(* CODESYS project mem_workflowlib.library
   Author: Ronny Walther
   Placeholder: MEM_WorkflowLib
   Title: MEM_WorkflowLib
   Version: 1.0.0.42
   Company: ME

Project tree, tasks and I/O mapping:
  libraries: Tc2_Standard, * (Beckhoff Automation GmbH); Tc2_System, * (Beckhoff Automation GmbH); Tc2_Utilities, * (Beckhoff Automation GmbH)
  AdsInterface/
    DUTs/
      data type eCmdProcessing
      data type eSendCmdProcessing
      data type TdocCmd
      data type TdocCmd2
      data type TdocRes
      data type TdocRes2
      data type TdwCmd2
      data type TdwRes2
      data type TwCmd
      data type TwCmd2
      data type TwRes
      data type TwRes2
      data type TxCmdRes
      data type TxCmdRes2
      data type TxCmdRes2Double
    function block FB_docCMD_Handler_Base [ST]: M_EnableCmd, M_ExecuteCommand, M_FinishCommand, M_Log, M_ReceiveCommand, P_EnabledInternally
    function block FB_SendAdsDocCmd_Base [ST]: M_EnableCmd, M_SendCmd, M_SetLocalData, P_CommandState, P_EnabledInternally
    function block FB_wCMD_docCMD_Handler_Base2 [ST]: A_LogResChanges, M_EnableCmd, M_ExecuteCommand, M_FinishCommand, M_Log, M_ReceiveCommand, P_EnabledInternally
    function block FB_wCMD_Handler_Base [ST]: M_EnableCmd, M_ExecuteCommand, M_FinishCommand, M_Log, M_ReceiveCommand, P_EnabledInternally
    global variables GVL_AdsInterface
    global variables GVL_AdsInterface_ERROR_IDS
    function InitializeAds_Incoming [ST]
    function InitializeAds_Outgoing [ST]
  DocManagement/
    DUTs/
      data type eDocPositionIndex
      data type sDocEvent
      data type sDocument
      data type ST_Document
      data type ST_Document_AdditionalData
      data type ST_Document_Path
      data type ST_Document_Position
      data type ST_Document_Processing
    program DocManagement [ST]: M_CheckDocsInPrevLocation, M_FindDoc, M_GetDocArrayInformation, M_GetDocInfoById, M_Initialize, M_InsertNewDoc, M_InsertNewDoc2, M_RedirectDoc, M_RemoveAllDocs, M_RemoveDoc, M_ResetDocMng, M_SethPath, M_SetReleased, P_iArraySize
    program DocManagement_Ext [ST]: M_CheckDocsInPrevLocation, M_FindDoc, M_GetDocArrayInformation, M_GetDocInfoById, M_Initialize, M_InsertNewDoc, M_RedirectDoc, M_RemoveAllDocs, M_RemoveDoc, M_ResetDocMng, M_SethPath, M_SetReleased, P_iArraySize
    global variables GVL_DocManagement
    global variables GVL_DocManagement_ERROR_IDS
  ErrorManagement/
    DUTs/
      data type E_ErrorLevels
      data type E_ErrorTypes
      data type eErrorHandlingMode
      data type eErrorHandlingMode_1
      data type eErrorNotificationMode
      data type eErrorNotificationMode_1
      data type eErrorTypes
      data type sErrorMsg
      data type sSystemError
      data type sSystemErrorEvent
      data type ST_ErrorMsg
      data type ST_SystemError
      data type ST_SystemErrorEvent
      data type tErrorConstant
    program ErrorManagement [ST]: M_GetErrorArrayInformation, M_GetErrorInfo, M_Initialize, M_InsertNewError, M_RemoveAllErrors, M_RemoveError, M_ResetSysErrorMng, M_SendAllErrorOnce, M_SendEvents, M_SendSingleError, P_bHaveAllErrorsBeenSentAtLeastOnce, P_ErrorNotificationMode, P_tEventIntervall, M_CreateEvent, M_CreateLogData
    program ErrorManagement_Ext [ST]: M_GetErrorArrayInformation, M_GetErrorInfo, M_Initialize, M_InsertNewError, M_RemoveAllErrors, M_RemoveError, M_ResetSysErrorMng, M_SendAllErrorOnce, M_SendEvents, M_SendSingleError, P_bHaveAllErrorsBeenSentAtLeastOnce, P_ErrorNotificationMode, P_tEventIntervall, M_CreateEvent, M_CreateLogData
    function block FB_ErrorHandler_Base [ST]: M_ExecuteHandling_Automatic, M_ExecuteHandling_Continue, M_ExecuteHandling_Repeat, M_IsHandlingModeAllowed, M_ResetFb, M_SetHandling, P_bHandlingAvailable, P_wAllowedHandlingModes
    global variables GVL_ErrorManagement
    global variables GVL_ErrorManagement_ERROR_IDS
  EventManager/
    DUTs/
      data type eValueEventNotificationModes
      data type sInfoEvent
      data type sInfoMessage
      data type sInfoMessageObject
      data type sValueEvent
      data type sValueEventNotificationParameter
      data type sValueEventObject
  Logging/
    DUTs/
      data type E_LogModes
      data type eLogLevel
      data type eLogPrgStates
      data type sLogMsg
      data type sLogMsgObject
    global variables GVL_Logging
    global variables GVL_Logging_ERROR_IDS
    program Logging [ST]: Debug, Error, Fatal, Info, M_Initialize, P_bAllDataWritten, P_bResetMaxLogBufferOccupancyInPct, P_iMaxFileSizeKB, P_iMaxLogBufferOccupancyInPct, P_LogLevel, P_LogPrgState, P_nCurLogBufferOccupancyInPct, Trace, Warn, M_CheckTargetAccess, M_CreateLogString, M_DeleteFile, M_GenerateFilepath, M_GetNextLogMsgtoWrite, M_InsertLog, M_RenameFile, M_UpdateCurFileSize, M_UpdateFilePath, M_UpdateSysTimeVar
  Standard/
    DUTs/
      data type E_RETVALUE
      data type eFbStates
      data type sMethodState
      data type ST_MethodState
      data type ST_MethodState_AdditionalData
      data type T_RETVALUE
    function Dec [ST]
    function block FB_MethodState [ST]: bBusy, bDone, bError, bTimeout, ErrorId, ErrorMsg, GoDoneState, GoNextState, GoSpecificState, GoStartState, iStateVar, Reset
    function block FB_MethodState_Ext [ST]: bBusy, bDone, bError, bTimeout, ErrorId, ErrorMsg, ErrorType, GoDoneState, GoNextState, GoSpecificState, GoStartState, iStateVar, Reset, T_RetVal
    function block FB_MethodState_Ext_Data [ST]
    global variables GVL
    function Inc [ST]
    function IsValidPtr [ST]
    interface ITF_MethodState: bBusy, bDone, bError, ErrorMsg, GoDoneState, GoNextState, GoSpecificState, GoStartState, iStateVar, Reset
    interface ITF_MethodState_Ext: bBusy, bDone, bError, ErrorMsg, GoDoneState, GoNextState, GoSpecificState, GoStartState, iStateVar, Reset
    function Scale [ST]
    function Switch [ST]
  Version/
    global variables Global_Version
  WorkstationFsm/
    DUTs/
      data type eSubState
      data type eWsOperationType
      data type eWsStates
      data type sWsConfiguration
    function block FB_WsFsm_Base [ST]: A_DoTransition, FB_init, M_ThrowError, M_ERROR_DO, M_PAST_HANDLING_DO, M_PAST_HANDLING_ENTRY, M_PAST_HANDLING_EXIT, M_PRE_HANDLING_DO, M_PRE_HANDLING_ENTRY, M_PRE_HANDLING_EXIT, M_FinishCycle, M_ResetWs, M_ResolveErrorState, M_StartNewCycle, P_bDocInWs, P_CurState, P_iDocId, P_pCurDoc, P_tWsProcTimeout, M_CYCLE_FINISHED_DO, M_CYCLE_FINISHED_ENTRY, M_CYCLE_FINISHED_EXIT, M_ERROR_ENTRY, M_ERROR_EXIT, M_IDLE_DO, M_IDLE_ENTRY, M_IDLE_EXIT, M_INIT_WS_DO, M_INIT_WS_ENTRY, M_INIT_WS_EXIT, M_MASTER_SYSTEM_PROCESSING_DO, M_MASTER_SYSTEM_PROCESSING_ENTRY, M_MASTER_SYSTEM_PROCESSING_EXIT, M_WS_PROCESSING_INTO_ERROR
    global variables GVL_Statemachine_ERROR_IDS
    function InitializeWsFsm_Base [ST]
    interface ITF_WsFsm: M_ERROR_DO, M_PAST_HANDLING_DO, M_PAST_HANDLING_ENTRY, M_PAST_HANDLING_EXIT, M_PRE_HANDLING_DO, M_PRE_HANDLING_ENTRY, M_PRE_HANDLING_EXIT
  00000000-0000-0000-0000-000000000000|ReleaseNotes.txt
  ReleaseNotes.txt
*)

// AdsInterface/DUTs/eCmdProcessing
{attribute 'qualified_only'}
TYPE eCmdProcessing :
(
	_UNDEFINED 			:= 0,
	_RECEIVING			:= 1,
	_WAITING_FOR_START	:= 2,
	_EXECUTING			:= 3,
	_ABORTING			:= 4,
	_FINISHING			:= 5
)UINT;
END_TYPE

// AdsInterface/DUTs/eSendCmdProcessing
{attribute 'qualified_only'}
TYPE eSendCmdProcessing :
(
	_UNDEFINED 	:= 0,
	_IDLE		:= 1,
	_SENDING	:= 2,
	_STARTING	:= 3,
	_EXECUTING	:= 4,
	_DONE		:= 5
)UINT;
END_TYPE

// AdsInterface/DUTs/TdocCmd
{attribute 'qualified_only'}
TYPE TdocCmd :
	STRUCT
		Control: 		WORD;					// 0 = stop, 1 = receive, 2 = start				
		Version: 		WORD;					// 0 = not defined, > 0 = version of the instruction	
		Reserved: 		WORD;
		ParaCount1:		BYTE;					// count of ParaData / byte                             		
		ParaTyp1:		BYTE;
		ParaData1:		DWORD;
		ParaCount2:		BYTE;					// count of ParaData / byte                             		
		ParaTyp2:		BYTE;
		ParaData2:		ARRAY [0..24] OF WORD;	// data									
	END_STRUCT
END_TYPE

// AdsInterface/DUTs/TdocCmd2
{attribute 'qualified_only'}
TYPE TdocCmd2 :
	STRUCT
		Control: 		WORD;					// 0 = stop, 1 = receive, 2 = start				
		Version: 		WORD;					// 0 = not defined, > 0 = version of the instruction
		CmdDataLengthIn8Byte:	BYTE;			// data lenth = const = 7 * 8 byte = 56 byte = 28 words
		ResDataLengthIn8Byte:	BYTE;			// data lenth = const = 7 * 8 byte = 56 byte = 28 words	
	
		//  rest 56 byte
		ParaCount1:		BYTE;					// count of ParaData / byte                             		
		ParaTyp1:		BYTE;
		ParaData1:		DWORD;
		ParaCount2:		BYTE;					// count of ParaData / byte                             		
		ParaTyp2:		BYTE;
		ParaData2:		ARRAY [0..23] OF WORD;	// data									
	END_STRUCT
END_TYPE

// AdsInterface/DUTs/TdocRes
{attribute 'qualified_only'}
TYPE TdocRes :
	STRUCT
		Status: 		WORD;					// 0 = not defined, 1 = received, 2 = aktive started, 3 = aktive aborting, 4 = finnished ok, 5 = finished stopped, 6 = finished error   
		Error: 			WORD;					// 0 = not defined, > 0 = error no
		ErrorComp: 		WORD;
		ParaCount1:		BYTE;					// count of ParaData / byte                             		
		ParaTyp1:		BYTE;
		ParaData1:		DWORD;
		ParaCount2:		BYTE;					// count of ParaData / byte                             		
		ParaTyp2:		BYTE;
		ParaData2:		ARRAY [0..24] OF WORD;	// data		
	END_STRUCT
END_TYPE

// AdsInterface/DUTs/TdocRes2
{attribute 'qualified_only'}
TYPE TdocRes2 :
	STRUCT
		Status: 		WORD;					// 0 = not defined, 1 = received, 2 = aktive started, 3 = aktive aborting, 4 = finnished ok, 5 = finished stopped, 6 = finished error   
		Error: 			WORD;					// 0 = not defined, > 0 = error no
		ErrorComp: 		WORD;
		
		//  rest 56 byte
		ParaCount1:		BYTE;					// count of ParaData / byte                             		
		ParaTyp1:		BYTE;
		ParaData1:		DWORD;
		ParaCount2:		BYTE;					// count of ParaData / byte                             		
		ParaTyp2:		BYTE;
		ParaData2:		ARRAY [0..23] OF WORD;	// data		
	END_STRUCT
END_TYPE

// AdsInterface/DUTs/TdwCmd2
{attribute 'qualified_only'}
TYPE TdwCmd2 :
	STRUCT
		Control: 				WORD;					// 0 = stop, 1 = receive, 2 = start				
		Version: 				WORD;					// 0 = not defined, > 0 = version of the instruction	
		CmdDataLengthIn8Byte:	BYTE;					// data lenth = const = 7 * 8 byte = 56 byte = 28 words
		ResDataLengthIn8Byte:	BYTE;					// data lenth = const = 7 * 8 byte = 56 byte = 28 words	
		
		//  rest 56 byte
		ParaCount1:				BYTE;					// count of ParaData / byte                             		
		ParaTyp1:				BYTE;		
		ParaData1:				ARRAY [0..12] OF DWORD;	// data
		ParaDummy1:				WORD;									
	END_STRUCT
END_TYPE

// AdsInterface/DUTs/TdwRes2
{attribute 'qualified_only'}
TYPE TdwRes2 :
	STRUCT
		Status: 		WORD;					// 0 = not defined, 1 = received, 2 = aktive started, 3 = aktive aborting, 4 = finnished ok, 5 = finished stopped, 6 = finished error   
												// 4 = finnished ok, 5 = finished stopped, 6 = finished error  
		Error: 			WORD;					// Unique Error ID, see GVL_Error_Constants
		ErrorComp: 		WORD;					// Unique Component ID, see GVL_Error_Constants
		
		//  rest 56 byte
		ParaCount1:		BYTE;					// count of ParaData / byte                             		
		ParaTyp1:		BYTE;
		ParaData1:		ARRAY [0..12] OF DWORD;	// parameter field
		ParaDummy1:		WORD;
	END_STRUCT
END_TYPE

// AdsInterface/DUTs/TwCmd
{attribute 'qualified_only'}
TYPE TwCmd :
	STRUCT
		Control: 		WORD;					// 0 = stop, 1 = receive, 2 = start				
		Version: 		WORD;					// 0 = not defined, > 0 = version of the instruction	
		Reserved: 		WORD;
		ParaCount:		BYTE;					// count of ParaData / byte                             		
		ParaTyp:		BYTE;
		ParaData:		ARRAY [0..27] OF WORD;	// data									
	END_STRUCT
END_TYPE

// AdsInterface/DUTs/TwCmd2
{attribute 'qualified_only'}
TYPE TwCmd2 :
	STRUCT
		Control: 				WORD;					// 0 = stop, 1 = receive, 2 = start				
		Version: 				WORD;					// 0 = not defined, > 0 = version of the instruction	
		CmdDataLengthIn8Byte:	BYTE;					// data lenth = const = 7 * 8 byte = 56 byte = 28 words
		ResDataLengthIn8Byte:	BYTE;					// data lenth = const = 7 * 8 byte = 56 byte = 28 words	
		
		//  rest 56 byte
		ParaCount1:				BYTE;					// count of ParaData / byte                             		
		ParaTyp1:				BYTE;		
		ParaData1:				ARRAY [0..26] OF WORD;	// data									
	END_STRUCT
END_TYPE

// AdsInterface/DUTs/TwRes
{attribute 'qualified_only'}
TYPE TwRes :
	STRUCT
		Status: 		WORD;					// 0 = not defined, 1 = received, 2 = aktive started, 3 = aktive aborting, 4 = finnished ok, 5 = finished stopped, 6 = finished error   
												// 4 = finnished ok, 5 = finished stopped, 6 = finished error  
		Error: 			WORD;					// Unique Error ID, see GVL_Error_Constants
		ErrorComp: 		WORD;					// Unique Component ID, see GVL_Error_Constants
		ParaCount:		BYTE;					// count of ParaData / byte                             		
		ParaTyp:		BYTE;
		ParaData:		ARRAY [0..27] OF WORD;	// parameter field
	END_STRUCT
END_TYPE

// AdsInterface/DUTs/TwRes2
{attribute 'qualified_only'}
TYPE TwRes2 :
	STRUCT
		Status: 		WORD;					// 0 = not defined, 1 = received, 2 = aktive started, 3 = aktive aborting, 4 = finnished ok, 5 = finished stopped, 6 = finished error   
												// 4 = finnished ok, 5 = finished stopped, 6 = finished error  
		Error: 			WORD;					// Unique Error ID, see GVL_Error_Constants
		ErrorComp: 		WORD;					// Unique Component ID, see GVL_Error_Constants
		
		//  rest 56 byte
		ParaCount1:		BYTE;					// count of ParaData / byte                             		
		ParaTyp1:		BYTE;
		ParaData1:		ARRAY [0..26] OF WORD;	// parameter field
	END_STRUCT
END_TYPE

// AdsInterface/DUTs/TxCmdRes
TYPE TxCmdRes :
	UNION
		wCmd: TwCmd;		// data of type word
		docCmd: TdocCmd;	// doc data type
		wRes: TwRes;		// data of type word
		docRes:	TdocRes;	// doc data type
	END_UNION
END_TYPE

// AdsInterface/DUTs/TxCmdRes2
TYPE TxCmdRes2 :
	UNION
		wCmd: TwCmd2;		// data of type word
		dwCmd: TdwCmd2;		// data of type dword
		docCmd: TdocCmd2;	// doc data type
		
		wRes: TwRes2;		// data of type word
		dwRes: TdwRes2;		// data of type dword
		docRes:	TdocRes2;	// doc data type
	END_UNION
END_TYPE

// AdsInterface/DUTs/TxCmdRes2Double
{attribute 'qualified_only'}
TYPE TxCmdRes2Double :
	STRUCT
		Cmd: TxCmdRes2;
		Res: TxCmdRes2;
	END_STRUCT
END_TYPE

// DocManagement/DUTs/eDocPositionIndex
TYPE eDocPositionIndex :
(
	UNDEFINED 	:= 0,
	POSITION_1 	:= 1,
	POSITION_2 	:= 2
)UINT;
END_TYPE

// DocManagement/DUTs/sDocEvent
//Event structure to send document tracking information without special request from host
//e.g. DocIn/ DocOut when entering/leaving a workstation and DocProcessStart when a doc is set to "UNRELEASED"
//Size: 6 Byte
TYPE sDocEvent :
	STRUCT
		DocID :				UDINT;	//Unique document id
		EventChangeFlag :	BOOL;	//assures that events ALWAYS differ from the previous one, not evaluated by host
	END_STRUCT
END_TYPE

// DocManagement/DUTs/sDocument
 
TYPE sDocument :
	STRUCT
		Free :					BOOL;	//0: Occupied, 1: Free
		ID :					UDINT;	//0: Document Identification (in the Machine)
		Module :				UINT;	//0: Invalid, 1: Modul 1, 2: Modul 2, 3: Modul 3
		Location :				UINT;	//0: Invalid, 1: RFID1, 2: RFID2, etc.
		Path :					UINT;	//Paths that the document could go through in the machine
		RedAtLocation :			UINT;	//0: No redirect, > 0: Location where document should be redirected
		RedToLocation :			UINT;	//0: No redirect, > 0: Location to where document should be redirected
		PositionIndex : 		UINT;	//Doc Position within a double usage. Only interesting if 2 different step sizes and 2 different layouts
		Released :				BOOL;	//0: Blocked, 1: Released (can be moved to next Location or picked up)
		bReleaseHandshakeActive: BOOL;	//Flag to switch release handshaking inside a non-virtual on or off
		Moving :				BOOL;	//0: Not Moving, 1: Moving
		bLockedBySps :			BOOL;	//FALSE: Doc can be modified by host, TRUE: Doc is locked by SPS and can not be modified by host
		Error :					BOOL;	//0: No Error, 1: Error
		//ErrorID :				WORD;	//ErrorID
	END_STRUCT
END_TYPE

// DocManagement/DUTs/ST_Document
 
TYPE ST_Document :
	STRUCT
		ID                      : UDINT;						//Unique document identification (in the Machine)

		stPosition 				: ST_Document_Position;			//Specifies the current position of the document inside the machine	
		stPath 					: ST_Document_Path; 			//Path of the document through the machine				
		stAdditionalData 		: ST_Document_AdditionalData;	//Various additional data
		stProcessing 			: ST_Document_Processing;		
		Free 					: BOOL;	//0: Occupied, 1: Free
	END_STRUCT
END_TYPE

// DocManagement/DUTs/ST_Document_AdditionalData
TYPE ST_Document_AdditionalData :
STRUCT
	DataString 	: STRING(GVL_DocManagement.MAX_INFO_TEXT_SIZE);
	DataField1	: LREAL;	//8bytes
	DataFiled2	: UDINT;	//4bytes
	DataField3	: UINT;		//2bytes
	DataField4 	: BYTE;		//1byte
END_STRUCT
END_TYPE

// DocManagement/DUTs/ST_Document_Path
TYPE ST_Document_Path :
STRUCT
		Path :					UINT;	//Paths that the document could go through in the machine
		RedAtLocation :			UINT;	//0: No redirect, > 0: Location where document should be redirected
		RedToLocation :			UINT;	//0: No redirect, > 0: Location to where document should be redirected
END_STRUCT
END_TYPE

// DocManagement/DUTs/ST_Document_Position
TYPE ST_Document_Position :
STRUCT		
		Module :				UINT;	//0: Invalid, 1: Modul 1, 2: Modul 2, 3: Modul 3
		Location :				UINT;	//0: Invalid, 1: RFID1, 2: RFID2, etc.
END_STRUCT
END_TYPE

// DocManagement/DUTs/ST_Document_Processing
TYPE ST_Document_Processing :
STRUCT
	bReleaseHandshakeActive	: BOOL;	//Flag to switch release handshaking inside a non-virtual on or off		
	Released 				: BOOL;	//0: Blocked, 1: Released (can be moved to next Location or picked up)	
	bLockedBySps 			: BOOL;	//FALSE: Doc can be modified by host, TRUE: Doc is locked by SPS and can not be modified by host
	Error 					: BOOL;	//FALSE: No Error, TRUE: Error
END_STRUCT
END_TYPE

// ErrorManagement/DUTs/E_ErrorLevels
{attribute 'qualified_only'}
TYPE E_ErrorLevels :
(
	_UNDEFINED 	:= 0,
	_WARNING	:= 1, 	//Machine continues running with some functionality deactivated eventually
	_ERROR		:= 2, 	//Machine shall be in ERROR state. Error can be solved by operator. A document reject could be possible
	_FATAL 		:= 3	//Machine shall be in ERROR state. Error can not be solved without major action. Could be a complete restart with all documents getting rejected
)UINT;
END_TYPE

// ErrorManagement/DUTs/E_ErrorTypes
{attribute 'qualified_only'}
TYPE E_ErrorTypes :
(
	SPS			:= 0, 	//firmware internal errors
	TWINCAT		:= 1 	//forwarded Beckhoff Twincat errors
)UINT;
END_TYPE

// ErrorManagement/DUTs/eErrorHandlingMode
{attribute 'qualified_only'}
TYPE eErrorHandlingMode :
(
	_NONE 		:= 0,
	_AUTOMATIC	:= 1,
	_REPEAT		:= 2,
	_CONTINUE	:= 3,
	_CANCEL		:= 4
)UINT;
END_TYPE

// ErrorManagement/DUTs/eErrorHandlingMode_1
{attribute 'qualified_only'}
TYPE eErrorHandlingMode_1 :
(
	_NONE 		:= 0,
	_AUTOMATIC	:= 1,
	_REPEAT		:= 2,
	_CONTINUE	:= 3,
	_CANCEL		:= 4
)UINT;
END_TYPE

// ErrorManagement/DUTs/eErrorNotificationMode
{attribute 'qualified_only'}
TYPE eErrorNotificationMode :
(
	UNDEFINED 							:= 0,
	SENDING_ERRORS_OFF					:= 1,
	SENDING_ERRORS_ONCE_IMMEDIATLY		:= 2,
	SENDING_ERRORS_ALWAYS_PERIODICALLY	:= 3
)UINT;
END_TYPE

// ErrorManagement/DUTs/eErrorNotificationMode_1
{attribute 'qualified_only'}
TYPE eErrorNotificationMode_1 :
(
	UNDEFINED 							:= 0,
	SENDING_ERRORS_OFF					:= 1,
	SENDING_ERRORS_ONCE_IMMEDIATLY		:= 2,
	SENDING_ERRORS_ALWAYS_PERIODICALLY	:= 3
)UINT;
END_TYPE

// ErrorManagement/DUTs/eErrorTypes
{attribute 'qualified_only'}
TYPE eErrorTypes :
(
	_UNDEFINED 	:= 0,
	_WARNING	:= 1, 	//Machine continues running with some functionality deactivated eventually
	_ERROR		:= 2, 	//Machine shall be in ERROR state. Error can be solved by operator. A document reject could be possible
	_FATAL 		:= 3	//Machine shall be in ERROR state. Error can not be solved without major action. Could be a complete restart with all documents getting rejected
)UINT;
END_TYPE

// ErrorManagement/DUTs/sErrorMsg
{attribute 'qualified_only'}
TYPE sErrorMsg : //to hold all SPS internal error messages
STRUCT
	//Categorization
		ErrorTyp : 		eErrorTypes;        //Undefined, Minor, Major, Fatal
	
	//Cause
		wModule : 		WORD := 1;				//Module no if redundant modules exist
		wComponent : 	WORD := 0;				//ID for each component
		wErrorNo : 		WORD := GVL.ERR_NO_ERROR;	//Error no (see GVL_Error_Constants)
		sFunctionName : STRING;					//name of (FSM) funtion which threw the error
	
	//Handling
		iRelatedDocId : UDINT := 0;
		pErrorHandler : POINTER TO FB_ErrorHandler_Base; //Pointer to specific error handler, if null pointer => no error handling
END_STRUCT
END_TYPE

// ErrorManagement/DUTs/sSystemError
{attribute 'qualified_only'}
TYPE sSystemError :
	STRUCT
		SysErrorMessageID :	UINT;		//Unique ID generated automatically by SysErrorMng. Helps to identify errors between SPS and host		
		ErrorMsg :			sErrorMsg;	//error msg structure
		bErrorWasSent :		BOOL;		//flag to indicate wether error was sent already or not
	END_STRUCT
END_TYPE

// ErrorManagement/DUTs/sSystemErrorEvent
//Event structure to send error information without special request from host
//Size: 18 Byte
{attribute 'qualified_only'}
TYPE sSystemErrorEvent :
	STRUCT
		iRelatedDocId : 		UDINT;			//rom error affected document, 0 = No doc affected
		
		SysErrorMessageID :		UINT;			//Unique ID generated automatically by SysErrorMng. Helps to identify errors between SPS and host
		
		ErrorTyp : 				eErrorTypes;	//Undefined, Minor, Major, Fatal		
		ErrorModuleId :			WORD;			//Machine module which holds the error reporting component	
		ErrorCompId :			WORD;			//Error reporting component
		ErrorId :				WORD;			//Unique error ID specifies the error happened

		AvailableHandlingModes:	WORD;			//Bits 0: none, 1:Automatic, 2:Repeat, 3: Continue
		EventChangeFlag:		BOOL;			//assures that events ALWAYS differ from the previous one, not evaluated by host
	END_STRUCT
END_TYPE

// ErrorManagement/DUTs/ST_ErrorMsg
{attribute 'qualified_only'}
TYPE ST_ErrorMsg : //to hold all SPS internal error messages
STRUCT
	//Categorization
		eErrorType : 		E_ErrorTypes; 
		eErrorLevel : 		E_ErrorLevels;        //Undefined, Minor, Major, Fatal
	
	//Cause
		wModule : 		WORD := 1;				//Module no if redundant modules exist
		wComponent : 	WORD := 0;				//ID for each component
		wErrorNo : 		WORD := GVL.ERR_NO_ERROR;	//Error no (see GVL_Error_Constants)
		sFunctionName : STRING;					//name of (FSM) funtion which threw the error
	
	//Handling
		iRelatedDocId : UDINT := 0;
		pErrorHandler : POINTER TO FB_ErrorHandler_Base; //Pointer to specific error handler, if null pointer => no error handling
END_STRUCT
END_TYPE

// ErrorManagement/DUTs/ST_SystemError
{attribute 'qualified_only'}
TYPE ST_SystemError :
	STRUCT
		SysErrorMessageID :	UINT;		//Unique ID generated automatically by SysErrorMng. Helps to identify errors between SPS and host		
		ErrorMsg :			ST_ErrorMsg;	//error msg structure
		bErrorWasSent :		BOOL;		//flag to indicate wether error was sent already or not
	END_STRUCT
END_TYPE

// ErrorManagement/DUTs/ST_SystemErrorEvent
//Event structure to send error information without special request from host
//Size: 18 Byte
{attribute 'qualified_only'}
TYPE ST_SystemErrorEvent :
	STRUCT
		iRelatedDocId : 		UDINT;			//rom error affected document, 0 = No doc affected
		
		SysErrorMessageID :		UINT;			//Unique ID generated automatically by SysErrorMng. Helps to identify errors between SPS and host
		
		ErrorTyp : 				E_ErrorLevels;	//Undefined, Minor, Major, Fatal		
		ErrorModuleId :			WORD;			//Machine module which holds the error reporting component	
		ErrorCompId :			WORD;			//Error reporting component
		ErrorId :				WORD;			//Unique error ID specifies the error happened

		AvailableHandlingModes:	WORD;			//Bits 0: none, 1:Automatic, 2:Repeat, 3: Continue
		EventChangeFlag:		BOOL;			//assures that events ALWAYS differ from the previous one, not evaluated by host
	END_STRUCT
END_TYPE

// ErrorManagement/DUTs/tErrorConstant
{attribute 'qualified_only'}
TYPE tErrorConstant : WORD (0..32767); END_TYPE
//Value is limited to 15bit because of ADS ME host connection DLL

// EventManager/DUTs/eValueEventNotificationModes
TYPE eValueEventNotificationModes :
(
	UNDEFINED 								:= 0,
	ON_CHANGE_ALWAYS						:= 1,
	ON_CHANGE_TIME_VALUE_DIFF_FROM_LAST		:= 2,
	ON_CHANGE_TIME_VALUE_DIFF_FROM_SPECIFIC	:= 3,
	ON_CHANGE_TIME							:= 4,
	TIME_CHANGE								:= 5
)UINT;
END_TYPE

// EventManager/DUTs/sInfoEvent
//Event structure to send general information without special request from host
//e.g. machine information, while performing some asynchrone action inside SPS
//Size: 6 Byte
TYPE sInfoEvent :
	STRUCT
		ComponentId :		WORD;	//Unique ID to identify the component the message came from
		InfoMessageId :		WORD;	//see GVL_Constants for pre-defined messages
		EventChangeFlag :	BOOL;	//assures that events ALWAYS differ from the previous one, not evaluated by host
	END_STRUCT
END_TYPE

// EventManager/DUTs/sInfoMessage
TYPE sInfoMessage :
STRUCT
	wComponentId :		WORD;	//Unique ID to identify the component the message came from
	wInfoMessageId :	WORD;	//see GVL_Constants for pre-defined messages
END_STRUCT
END_TYPE

// EventManager/DUTs/sInfoMessageObject
TYPE sInfoMessageObject :
STRUCT
	bEventIsValid	: BOOL;
	InfoMessage 	: sInfoMessage;
END_STRUCT
END_TYPE

// EventManager/DUTs/sValueEvent
TYPE sValueEvent : 
	STRUCT
		Value 			: WORD; //event specific value
		EventChangeFlag : BOOL;	//assures that events ALWAYS differ from the previous one, not evaluated by host
		 {attribute 'hide'}
		_reserved1 : USINT;
	END_STRUCT
END_TYPE

// EventManager/DUTs/sValueEventNotificationParameter
TYPE sValueEventNotificationParameter :
STRUCT
	NotificationMode 	: eValueEventNotificationModes;	//notification mode
	tSendInterval 		: TIME;							//Minimum send interval 
	iValueDiff			: UINT;							//trigger tolerance in Modes: ON_CHANGE_TIME_VALUE_DIFF_FROM_LAST and ON_CHANGE_TIME_VALUE_DIFF_FROM_SPECIFIC
	iSpecificRefValue	: UINT;							//reference value to be compared to in Mode: ON_CHANGE_TIME_VALUE_DIFF_FROM_SPECIFIC
END_STRUCT
END_TYPE

// EventManager/DUTs/sValueEventObject
TYPE sValueEventObject :
STRUCT
	bEventIsValid			: BOOL;
	strEventName			: STRING;
	pInternallyLinkedValue	: POINTER TO UINT;	
	pEvent 					: POINTER TO sValueEvent;
	EventParameter			: sValueEventNotificationParameter;
	tTimer					: TON;
END_STRUCT
END_TYPE

// Logging/DUTs/E_LogModes
{attribute 'qualified_only'}
{attribute 'strict'}
TYPE E_LogModes :
(
	KeepAllFiles 	:= 0,
	KeepTwoFiles 	:= 1
);
END_TYPE

// Logging/DUTs/eLogLevel
// ALL → TRACE → DEBUG → INFO → WARN → ERROR → FATAL → OFF.
{attribute 'qualified_only'}
TYPE eLogLevel :
(
	OFF			:= 0,	
//Log levels	
	FATAL		:= 1,
	ERROR 		:= 2,
	WARN 		:= 3,
	INFO 		:= 4,	
	DEBUG 		:= 5,
	TRACE		:= 6,	
	ALL			:= 7
)UINT;
END_TYPE

// Logging/DUTs/eLogPrgStates
{attribute 'qualified_only'}
TYPE eLogPrgStates :
(
	LOG_INITIALIZING 	:= 0,
	LOG_STAND_BY		:= 1,
	LOG_OPENING_FILE	:= 2,
	LOG_WRITING_FILE	:= 3,
	LOG_CLOSING_FILE	:= 4,
	LOG_ERROR			:= 5
)UINT;
END_TYPE

// Logging/DUTs/sLogMsg
{attribute 'qualified_only'}
TYPE sLogMsg :
	STRUCT
		LogLevel 			: eLogLevel;
		sCallFunctionName 	: STRING;			//name of (FSM) funtion which threw the error		
		sLogMessage 		: STRING(255);	
	END_STRUCT
END_TYPE

// Logging/DUTs/sLogMsgObject
{attribute 'hide'}
{attribute 'qualified_only'}
TYPE sLogMsgObject :
	STRUCT
		bIsValidMsg	: BOOL;
		iLogMsgId 	: UDINT;			//Unique ID generated automatically by SysErrorMng. Helps to identify errors between SPS and host
		sTimeStamp 	: STRING;
		LogMsg 		: sLogMsg;
	END_STRUCT
END_TYPE

// Standard/DUTs/E_RETVALUE
//{attribute 'qualified_only'}
//{attribute 'strict'}
TYPE E_RETVALUE :
(
	eOK 	 := 1,
	eBUSY 	 := 0,
	eNOK 	 := -1	
)INT;
END_TYPE

// Standard/DUTs/eFbStates
{attribute 'qualified_only'}
TYPE eFbStates : //Types to structure FB state machines
(
	_ENTRY 			:= 0,
	_OFF			:= 1,
	_POWERING_ON	:= 2,
	_INITIALIZING	:= 3,
	_IDLE			:= 4,
	_RUNNING		:= 5,
	_POWERING_OFF	:= 6,
	_ERROR			:= 7,	 
	_EXIT			:= 8
)uint;
END_TYPE

// Standard/DUTs/sMethodState
{attribute 'qualified_only'}
TYPE sMethodState :
STRUCT
	//Status flags
		bDone 		: BOOL;
		bError 		: BOOL;
		bBusy		: BOOL;
		(*
	//signals, if the corresponding status flag just changed (rising or falling edge)
		bDoneEdge,
		bErrorEdge,
		bBusyEdge	: BOOL;
		*)
	iStateVar	: UINT;
	ErrorMsg 	: sErrorMsg;
END_STRUCT
END_TYPE

// Standard/DUTs/ST_MethodState
{attribute 'qualified_only'}
TYPE ST_MethodState :
STRUCT
	//Status flags
		bDone 		: BOOL;
		bError 		: BOOL;
		bBusy		: BOOL;
		(*
	//signals, if the corresponding status flag just changed (rising or falling edge)
		bDoneEdge,
		bErrorEdge,
		bBusyEdge	: BOOL;
		*)
		iStateVar	: UINT;
		ErrorMsg 	: ST_ErrorMsg;
END_STRUCT
END_TYPE

// Standard/DUTs/ST_MethodState_AdditionalData
TYPE ST_MethodState_AdditionalData :
STRUCT
	DataString 	: STRING(GVL_DocManagement.MAX_INFO_TEXT_SIZE);
	DataField1	: LREAL;	//8bytes
	DataFiled2	: UDINT;	//4bytes
	DataField3	: UINT;		//2bytes
	DataField4 	: BYTE;		//1byte
END_STRUCT
END_TYPE

// Standard/DUTs/T_RETVALUE
TYPE T_RETVALUE : E_RETVALUE; END_TYPE

// WorkstationFsm/DUTs/eSubState
{attribute 'qualified_only'}
{attribute 'strict'}
TYPE eSubState :
(
	UNDEFINED 	:= 0,
	STATE_ENTRY	:= 1,
	STATE_DO	:= 2,
	STATE_EXIT	:= 3	
);
END_TYPE

// WorkstationFsm/DUTs/eWsOperationType
TYPE eWsOperationType :
(
	_UNDEFINED 				:= 0,
	_STEP_BY_STEP			:= 1,	//workstation cycling is controlled step by step
	_CONTINOUS_BY_TRIGGER	:= 2	//workstation cycling is triggered by a external s signal
)UINT;
END_TYPE

// WorkstationFsm/DUTs/eWsStates
TYPE eWsStates : //Possible Workstation states inside FB_WsFsm
(
	UNDEFINED 					:= 0,
	INIT_WS						:= 1,
	IDLE						:= 2,	//WS ready to be startet
	WS_PROCESSING				:= 3,	//WS running (including Master system processing)
	PRE_HANDLING				:= 4,	//optional code can be processed here
	MASTER_SYSTEM_PROCESSING	:= 5,	//Master system is processing the document
	PAST_HANDLING				:= 6,	//optional code can be processed here
	ERROR						:= 7,	//Ws in error
	CYCLE_FINISHED				:= 8	//Cycle ready to be finished
)UINT;
END_TYPE

// WorkstationFsm/DUTs/sWsConfiguration
TYPE sWsConfiguration :
STRUCT
	iWsNum : 					UINT;
	iRelDocNum :				UINT;	//Distance between previous and this WS in mm - 0 is OFF
	iLocation :					UINT;		
	bVirtualWs : 				BOOL;
	tWsProcessingTimeout :		TIME;	//Timeout for composite state WsProcessing
	OperationType: 				eWsOperationType;

//Doc events	
	pEvt_DocIn, 
	pEvt_DocProcessStart,
	pEvt_DocOut : 				POINTER TO sDocEvent;
	bEvt_DocIn_WasSet, 									//DocIn event set status
	pEvt_DocProcessStart_WasSet,						//DocProcessStart event set status
	pEvt_DocOut_wasSet 				: BOOL := FALSE;	//DocOut event set status
	
	wCompId : 					WORD;	
	//Document will be unlocked when method M_FinishCycle is called. 
	//Flag shall be set to TRUE, if Ws is the last WS to enable the host to remove the doc from the buffer
	bUnlockDocAtFinishing : BOOL; 
END_STRUCT
END_TYPE

// AdsInterface/GVL_AdsInterface
{attribute 'hide'}
{attribute 'qualified_only'}
VAR_GLOBAL
	wCompId_IncomingAds,
	wCompId_OutgoingAds 		: tErrorConstant	:= 0;
	
	wErrorIdOffset_IncomingAds,
 	wErrorIdOffset_OutgoingAds	: tErrorConstant	:= 0;
	
	bLoggingOnOff_IncomingAds,
	bLoggingOnOff_OutgoingAds 	: BOOL				:= FALSE;
END_VAR

// AdsInterface/GVL_AdsInterface_ERROR_IDS
{attribute 'qualified_only'}
VAR_GLOBAL CONSTANT	
	ERR_ITF_INCOMING_COMMAND_HAS_WRONG_VERSION :							tErrorConstant := 1;
	ERR_ITF_INCOMING_COMMAND_HAS_WRONG_PARAMETER_COUNT :					tErrorConstant := 2;
	ERR_ITF_INCOMING_COMMAND_HAS_WRONG_PARAMETER_TYP :						tErrorConstant := 3;
	ERR_ITF_INCOMING_COMMAND_IS_BLOCKED :									tErrorConstant := 4;
	ERR_ITF_COMMAND_CAN_NOT_BE_ENABLED_THUS_INTERNALLY_DISABLED:			tErrorConstant := 5;
	ERR_ITF_COMMAND_CAN_NOT_BE_ENABLED_THUS_EXTERNALLY_DISABLED:			tErrorConstant := 6;
	ERR_ITF_WRONG_COMMAND_DATA:												tErrorConstant := 7;
	ERR_ITF_COMMAND_EXECUTION_TIMEOUT:										tErrorConstant := 8;
	ERR_ITF_INCOMING_COMMAND_HAS_WRONG_COMMAND_DATA_SIZE:					tErrorConstant := 9;
	ERR_ITF_INCOMING_COMMAND_HAS_WRONG_RESULT_DATA_SIZE:					tErrorConstant := 10;
	
	ERR_ITF_COMMAND_WAS_ABORTED_BY_HOST_DURING_EXECUTION:					tErrorConstant := 15;

	//ADS Sending errors
	ERR_ITF_WRONG_FB_STATE_TO_SEND_COMMAND :								tErrorConstant := 50;
	
END_VAR

// DocManagement/GVL_DocManagement
{attribute 'qualified_only'}
{attribute 'hide'}
VAR_GLOBAL
	wCompId 					: tErrorConstant	:= 0;
	wErrorIdOffset 				: tErrorConstant	:= 0;
END_VAR
VAR_GLOBAL CONSTANT
	MAX_INFO_TEXT_SIZE 			: UINT 				:= 50; 
END_VAR

// DocManagement/GVL_DocManagement_ERROR_IDS
{attribute 'qualified_only'}
VAR_GLOBAL CONSTANT
	
	ERR_DOC_ID_NOT_FOUND :													tErrorConstant := 2;
	ERR_DOC_ARRAY_FULL : 													tErrorConstant := 3;
	ERR_DOC_CAN_NOT_BE_INSERTED_THUS_DOC_ID_EXISTENT_ALREADY :				tErrorConstant := 4;
	ERR_DOC_CAN_NOT_BE_INSERTED_THUS_ARRAY_FULL :							tErrorConstant := 5;
	
	ERR_DOC_ID_ZERO_INVALID :												tErrorConstant := 10;	
	ERR_DOC_NUMBER_ZERO_INVALID :											tErrorConstant := 12;	
	ERR_DOC_NUMBER_HIGHER_THAN_ARRAY_SIZE :									tErrorConstant := 13;
	ERR_DOC_NUMBER_DOES_NOT_EXIST :											tErrorConstant := 14;
	ERR_DOC_ID_DOES_NOT_EXIST :												tErrorConstant := 15;
	ERR_DOC_ID_TO_BE_INSERTED_NOT_HIGHER_THAN_EXISTING_IDS :				tErrorConstant := 16;
	ERR_DOC_CAN_NOT_BE_REMOVED_THUS_LOCKED_BY_SPS :							tErrorConstant := 17;
	ERR_NOT_ALL_DOCS_COULD_BE_REMOVED_THUS_LOCKED_BY_SPS :					tErrorConstant := 18;
	ERR_DOC_CAN_NOT_BE_RELEASED_THUS_NOT_UNRELEASED :						tErrorConstant := 19;

	//Doc handover
	ERR_HANDOVER_DOC_COULD_NOT_BE_STARTED_THUS_LOCATION_INVALID :			tErrorConstant := 50;
	ERR_DOC_HANDOVER_COULD_NOT_BE_STARTED_THUS_DOC_POINTER_INVALID :		tErrorConstant := 51;
	ERR_HANDOVER_DOC_COULD_NOT_BE_FINISHED_THUS_WRONG_STATE :				tErrorConstant := 52;
	ERR_DOC_HANDOVER_COULD_NOT_BE_FINISHED_THUS_DOC_POINTER_INVALID :		tErrorConstant := 53;
END_VAR

// ErrorManagement/GVL_ErrorManagement
{attribute 'hide'}
{attribute 'qualified_only'}
VAR_GLOBAL
	wCompId 		: tErrorConstant	:= 0;
	wErrorIdOffset 	: tErrorConstant	:= 0;
	bLoggingOnOff 	: BOOL				:= FALSE;
	pEvt 			: POINTER TO sSystemErrorEvent := ADR(cDUMMY_EVENT); //Just here for compatibility in Errormanagement.prg
	
//ErrorManagement_Ext.prg only
	pEvt_SpsError		: POINTER TO ST_SystemErrorEvent := ADR(cDUMMY_EVENT_EXT);
	pEvt_TwincatError	: POINTER TO ST_SystemErrorEvent := ADR(cDUMMY_EVENT_EXT);
END_VAR
VAR_GLOBAL CONSTANT
	cDUMMY_EVENT 		: sSystemErrorEvent := (SysErrorMessageID := 0);
	cDUMMY_EVENT_EXT	: ST_SystemErrorEvent := (SysErrorMessageID := 0);
END_VAR

// ErrorManagement/GVL_ErrorManagement_ERROR_IDS
{attribute 'qualified_only'}
VAR_GLOBAL CONSTANT	
	ERR_ERROR_ID_NOT_FOUND :												tErrorConstant := 1;
	ERR_ERROR_ID_ZERO_INVALID :												tErrorConstant := 2;
	ERR_ERROR_ARRAY_FULL :													tErrorConstant := 3;
	
	ERR_SEND_ERRORS_ONCE_NOT_POSSIBLE_THUS_PERIODIC_SENDING_ACTIVATED :		tErrorConstant := 10;
	
	ERR_FSM_INVALID_ERROR_HANDLER_POINTER:									tErrorConstant := 20;
	ERR_FSM_NO_ERROR_HANDLING_AVAILABLE_INSIDE_HANDLER:						tErrorConstant := 21;
	ERR_FSM_PRE_SET_HANDLER_ERRORID_DIFFERS:								tErrorConstant := 22;
	ERR_FSM_ERROR_HANDLING_MODE_NOT_ALLOWED:								tErrorConstant := 23;	
END_VAR

// Logging/GVL_Logging
{attribute 'qualified_only'}
{attribute 'hide'}
VAR_GLOBAL
	wCompId 					: tErrorConstant	:= 0;
	wErrorIdOffset 				: tErrorConstant	:= 0;
	DEST_AMS_NET_ID 			: T_AmsNetId 		:= '';
	FILE_DESTINATION_DIRECTORY  : STRING 			:= 'C:\';
	FILE_NAME_PREFIX  			: STRING(20) 		:= 'SPS_LOG'; 
	FILE_NAME_EXT_OLD			: STRING(5)			:= 'OLD';
	eLogMode 					: E_LogModes 		:= E_LogModes.KeepAllFiles;
END_VAR

// Logging/GVL_Logging_ERROR_IDS
{attribute 'qualified_only'}
VAR_GLOBAL CONSTANT
	ERR_STRING_COULD_NOT_BE_WRITTEN_TO_THE_OPENED_LOG_FILE :	tErrorConstant := 1; //the log string could not be written to the log file
	ERR_LOG_FILE_COULD_NOT_BE_CLOSED :							tErrorConstant := 2; //the log file could not be closed
	ERR_LOG_FILE_TARGET_NOT_FOUND :								tErrorConstant := 3; //the target (PC) could not be found. Please check AmsNetId!
	ERR_LOG_FILE_COULD_NOT_BE_OPENED_OR_CREATED :				tErrorConstant := 4; //the log file could not be oppened or created. Please check file permissions on target (PC)!
END_VAR

// Standard/GVL
{attribute 'qualified_only'}
VAR_GLOBAL CONSTANT
	ERR_NO_ERROR : 												tErrorConstant := 0; //No error	
END_VAR

// Version/Global_Version
{attribute 'TcGenerated'}
{attribute 'no-analysis'}
{attribute 'linkalways'}
// This function has been automatically generated from the project information.
VAR_GLOBAL CONSTANT
	{attribute 'const_non_replaced'}
	stLibVersion_MEM_WorkflowLib : ST_LibVersion := (iMajor := 1, iMinor := 0, iBuild := 0, iRevision := 42, nFlags := 0, sVersion := '1.0.0.42');
END_VAR

// WorkstationFsm/GVL_Statemachine_ERROR_IDS
{attribute 'qualified_only'}
VAR_GLOBAL
	iErrorOffset 	: tErrorConstant 	:= 16000;
	bLoggingOnOff 	: BOOL				:= FALSE;
END_VAR
VAR_GLOBAL CONSTANT
	ERR_FSM_INVALID_WS_POINTER : 											tErrorConstant := 1;
	ERR_FSM_INVALID_DOC_POINTER : 											tErrorConstant := 2;	
	ERR_FSM_WS_IN_ERROR_STATE : 											tErrorConstant := 3;
	ERR_FSM_WS_IN_WRONG_STATE : 											tErrorConstant := 4;	
	ERR_FSM_WRONG_STATE_TO_FINISH_CYCLE : 									tErrorConstant := 5;
	ERR_FSM_WRONG_STATE_TO_START_NEW_CYCLE : 								tErrorConstant := 6;	
	ERR_FSM_WRONG_LOCATION_OF_NEW_DOC : 									tErrorConstant := 7;
	ERR_FSM_WRONG_INPUT_PARAMETER :											tErrorConstant := 8;		
	ERR_FSM_WS_PROCESSING_TIMEOUT :											tErrorConstant := 9;	
	ERR_FSM_WS_PROCESSING_HANDLING_ERROR : 									tErrorConstant := 10;	
	ERR_FSM_DOC_PROCESS_START_EVENT_NOT_SET :								tErrorConstant := 11;	
	ERR_FSM_WORKSTATION_ERROR_CAN_NOT_BE_RESOLVED : 						tErrorConstant := 12;
END_VAR

// AdsInterface/FB_docCMD_Handler_Base
//Author: 				Walther Ronny
//Version:				1.3
//Last change:			25.05.16
//See Release notes at the bottom
//{attribute 'hide_all_locals'}
{attribute 'reflection'}
FUNCTION_BLOCK PUBLIC FB_docCMD_Handler_Base				//Base Fb for handling of ADS communication of type TwRes and TwCmd
VAR_OUTPUT
    {attribute 'instance-path'}
    {attribute 'no_init'}
    sPath  : STRING;
	
END_VAR 
VAR_INPUT		
	Instanz: BYTE; 										//Instanz counter 
	pCmd : POINTER TO TxCmdRes;							//Pointer to incomming command structure from host
	pRes : POINTER TO TxCmdRes;							//Pointer to outgoing result structure from SPS
END_VAR
VAR
	wCompId : WORD;		//Component ID
//Command configuration which has to be set by instantiated Fb - 	MUST !
	wVersion : 				WORD := 0;	//Expected version of incomming command
	iParTyp1: 				BYTE := 0;	//Expected parameter type of incomming command, PAR_TYPE_REGARDLESS will switch test off
	iParCount1 : 			BYTE := 0;	//Expected parameter count of incomming command
	iParTyp2 : 				BYTE := 0;	//Expected parameter type of incomming command, PAR_TYPE_REGARDLESS will switch test off
	iParCount2 : 			BYTE := 0;	//Expected parameter count of incomming command
	
//Command configuration which can be set by instantiated Fb - 	OPTIONALLY !
	bAbortionAllowed : 		BOOL := FALSE;					//if yes, abortion from host is allowed all the time
	tExecutionTimeout : 	TIME := ADS_EXECUTION_TIMEOUT; 	//Timeout while Execution running. T#0s equals off
	strInstanceName :		STRING(40);								//Name of instance of that base class (used only for logging purposes)
//Flag to indicate that the derived method "M_ExecuteCommand()" finished	
	bExecutionDone : BOOL := FALSE;	//flag to indicate that derived Execution is done				

//This variable can be used to hold the state of the derived M_ExecuteCommand() 
	iHelpState : UINT := 0;	//optional help variable to create a statemachine inside derive M_ExecuteCommand()
	
//Local Command and result structure objects - Will be read and written by base Fb and derived "M_ExecuteCommand()" method
	localRes: TdocRes;
	localCmd: TdocCmd;	
	
//Internal variables of base Fb - DO NOT CHANGE!	
	bCmdEnabledByExtern,								//Command is enabled/disabled  externally (by MainFSM)
	bCmdEnabledByIntern : 	BOOL:= TRUE;				//Command is enabled/disabled  internally during execution
		
	eState: eCmdProcessing := eCmdProcessing._RECEIVING;	//Current internal state of the base Fb		
	TimerExecutionTimeout : ton;						// Timer for Execution timeout
END_VAR
VAR CONSTANT
	//Command parameter types
	PAR_TYPE_REGARDLESS :		BYTE := 0;		//if this type is set, the parameter type will be not checked
	PAR_TYPE_ANSICHAR : 		BYTE := 16#41; //8bit
	PAR_TYPE_BYTE : 			BYTE := 16#42; //8bit
	PAR_TYPE_WIDECHAR : 		BYTE := 16#43; //16bit
	PAR_TYPE_FLOAT : 			BYTE := 16#44; //64bit	
	PAR_TYPE_SHORTINT : 		BYTE := 16#53; //8bit	
	PAR_TYPE_SMALLINT : 		BYTE := 16#4D; //16bit
	PAR_TYPE_LONGINT : 			BYTE := 16#49; //32bit
	PAR_TYPE_LONGWORD : 		BYTE := 16#4C; //32bit
	PAR_TYPE_WORD : 			BYTE := 16#57; //16bit
	PAR_TYPE_BIT : 				BYTE := 16#58;
	
	ADS_EXECUTION_TIMEOUT :		TIME := T#30S;		//Timeout while derived Execution method is executed. T#0S equals OFF

		// command
	cAbort:						WORD := 0;			// command abort				
	cRcv:						WORD := 1;			// command receive				
	cExec:						WORD := 2;			// command start				
	// result
	cIdle: 						WORD := 0;      	// not  defined					
	cRcvd:						WORD := 1;      	// command received 			
	cActive:					WORD := 2;			// command active started 		
	cFinOk:						WORD := 4;			// command finished ok			
	cFinAbrtd:					WORD := 5;			// command aborted				
	cFinErr:					WORD := 6;			// command finished error		
END_VAR

(*
Release notes:
1.0 Initial version. Copy from FB_wCMD_Handler_Base
1.1 Walther Ronny, 22.02.16
	- Bug M_ReceiveCommand PARTYP_REGARDLESS fixed
1.3 Walther Ronny, 25.05.16
	- Variable strInstanceName added
	- Method M_Log() added
	- Logging added
*)

//Create local copy of received command struct
	localCmd := pCmd^.docCmd;

CASE eState OF
	
	eCmdProcessing._RECEIVING: 	//Receiving command
	
				//Check id, thus it might have been changed
					wCompId := GVL_AdsInterface.wCompId_IncomingAds;
				
				M_ReceiveCommand();
				
				IF localRes.Status = cRcvd THEN //was something received?	

					//Log data
						M_Log(	LogLevel 	:= eLogLevel.TRACE, 
								strMethod 	:= 'FB_docCMD_Handler_Base',
								strLogMsg 	:= '|ADS - command received from host');	
		
					eState := eCmdProcessing._WAITING_FOR_START;
					
				END_IF
				
	eCmdProcessing._WAITING_FOR_START:	//Waiting for Start from Host
	
				IF localCmd.Control = cExec THEN //check if the command was started by the host
					//Log data
						M_Log(	LogLevel 	:= eLogLevel.TRACE, 
								strMethod 	:= 'FB_docCMD_Handler_Base',
								strLogMsg 	:= '|ADS - command started by host');	
								
					IF localRes.Error = GVL.ERR_NO_ERROR THEN //Check if an error during receiving ocurred
						//Reset variables for derived "M_ExecuteCommand()" method	
							bExecutionDone := FALSE;
							iHelpState := 0;	
						
						localRes.Status := cActive;					
						eState := eCmdProcessing._EXECUTING;
						
						//start timeout timer
							TimerExecutionTimeout(IN := TRUE, PT := tExecutionTimeout);
					ELSE						
						eState := eCmdProcessing._FINISHING;
						
					END_IF
					
				END_IF
					
					
	eCmdProcessing._EXECUTING:	//Executing command
			
				IF bExecutionDone THEN //flag will be set by derived method if execution done									
					eState := eCmdProcessing._FINISHING; 
					
				ELSIF TimerExecutionTimeout.Q AND tExecutionTimeout <> T#0S THEN
					localRes.Error := GVL_AdsInterface_ERROR_IDS.ERR_ITF_COMMAND_EXECUTION_TIMEOUT + GVL_AdsInterface.wErrorIdOffset_IncomingAds;
					
					eState := eCmdProcessing._FINISHING; 			
					
				ELSE //derived method will be executed
					M_ExecuteCommand();
						
				END_IF
	
		
	eCmdProcessing._FINISHING: //Finishing Command
		
				M_FinishCommand();
				
				//reset timer
					TimerExecutionTimeout.IN := FALSE;
				
				
	eCmdProcessing._ABORTING: //Aborting Command
				
				eState := eCmdProcessing._FINISHING; 
				
END_CASE

//check if aborted by host and command configured "bAbortionAllowed
//Note: 	Thus abortion is possible all the time the execution could be interuppted at an unsafe state!
//			Preferable abortion should be allowed only for service commands which a triggered manually from an operator.
	IF localCmd.Control = cAbort AND bAbortionAllowed 
		AND eState <> eCmdProcessing._ABORTING 		//Not allowed cause aborting already active
		AND eState <> eCmdProcessing._FINISHING 	//Not allowed cause command is finishing anyway
		AND eState <> eCmdProcessing._RECEIVING		//Not allowed cause command have not been started yet
		THEN 
			
			IF eState = eCmdProcessing._EXECUTING THEN  //cause eventually leaving unsafe state, throw error
				localRes.Error := GVL_AdsInterface_ERROR_IDS.ERR_ITF_COMMAND_WAS_ABORTED_BY_HOST_DURING_EXECUTION + GVL_AdsInterface.wErrorIdOffset_IncomingAds;
				
			END_IF
			
			eState := eCmdProcessing._ABORTING;
			
	END_IF

TimerExecutionTimeout();

pRes^.docRes := localRes;

METHOD PUBLIC FINAL M_EnableCmd
VAR_INPUT
	bEnable : BOOL := FALSE; //TRUE = Command is enabled, FALSE = Command i disabled
END_VAR
bCmdEnabledByExtern := bEnable;
END_METHOD

METHOD public M_ExecuteCommand // to be derived and customized....
// to be derived and customized....



//To DO`s of the derived Method:
 
//1. Check Data for correctness
//2. set optional result data 
//3. iHelpState vaiable can be used
//4. if an Error occured localRes.Error and localRes.ErrorComp has to be set!
//5. at last the "bExecutionDone" flag has to be set. This will start the transition to the M_FinishCommand Method inside the base FB.

//Note: the execution time is monitored by a base Fb timer. Therefore a timeout may occur. This behavior is configurable.
END_METHOD

METHOD PRIVATE FINAL M_FinishCommand
VAR
	strLogMsg : STRING;
END_VAR
IF localCmd.Control = cAbort AND bAbortionAllowed THEN		//Command was aborted by host
	localRes.Status := cFinAbrtd;

ELSIF localRes.Error = GVL.ERR_NO_ERROR THEN					//executed without error
	localRes.Status := cFinOk;
	
	//Log data
		M_Log(	LogLevel 	:= eLogLevel.TRACE, 
				strMethod 	:= 'M_FinishCommand',
				strLogMsg 	:= '|ADS - command finished successfully by SPS');	
				
ELSE
	localRes.Status := cFinErr;								//executed with error
	//Log data
		strLogMsg := CONCAT('|ADS - command finished faulty by SPS with ErrorId: ', WORD_TO_STRING(localRes.Error));
	
		M_Log(	LogLevel 	:= eLogLevel.TRACE, 
				strMethod 	:= 'M_FinishCommand',
				strLogMsg 	:= strLogMsg);				
END_IF

bCmdEnabledByIntern := TRUE;
eState := eCmdProcessing._RECEIVING;
END_METHOD

METHOD PROTECTED FINAL M_Log
VAR_INPUT
	strMethod 	: STRING(40);
	strLogMsg 	: STRING;
	LogLevel 	: eLogLevel;
END_VAR
VAR
	strCaller : STRING := 'FB_wCMD_Handler_Base.';
END_VAR
IF NOT GVL_AdsInterface.bLoggingOnOff_IncomingAds THEN 
	RETURN;
END_IF

strCaller := CONCAT(strInstanceName, '.');
strCaller := CONCAT(strCaller, strMethod);

//If Logging.prg is not available in project or to deactivate logging completely, just comment the following line out!
	Logging.Debug(strCaller, strLogMsg);
END_METHOD

METHOD PRIVATE FINAL M_ReceiveCommand
IF localCmd.Control = cRcv THEN

	//Delete result structure variable
		MEMSET(destaddr := ADR(localRes), fillbyte:=0, n:= SIZEOF(localRes));
		localRes.ErrorComp 	:= wCompId;
		localres.Error 		:= GVL.ERR_NO_ERROR;
		
	//Set result struct to state RECEIVED even if there could be errors
		localRes.Status := cRcvd;
	
	//Check if command is currently blocked
	IF bCmdEnabledByExtern AND bCmdEnabledByIntern THEN
		bCmdEnabledByIntern := FALSE;
		
	ELSIF NOT bCmdEnabledByIntern THEN		
		localRes.Error := GVL_AdsInterface_ERROR_IDS.ERR_ITF_COMMAND_CAN_NOT_BE_ENABLED_THUS_INTERNALLY_DISABLED + GVL_AdsInterface.wErrorIdOffset_IncomingAds;
		
	ELSIF NOT bCmdEnabledByExtern THEN
		localRes.Error := GVL_AdsInterface_ERROR_IDS.ERR_ITF_COMMAND_CAN_NOT_BE_ENABLED_THUS_EXTERNALLY_DISABLED + GVL_AdsInterface.wErrorIdOffset_IncomingAds;
		
	ELSE
		localRes.Error := GVL_AdsInterface_ERROR_IDS.ERR_ITF_INCOMING_COMMAND_IS_BLOCKED + GVL_AdsInterface.wErrorIdOffset_IncomingAds;
		
	END_IF
	
	//Check incomming command parameter for correctness
		IF localCmd.Version 	<> wVersion 			THEN localRes.Error := GVL_AdsInterface_ERROR_IDS.ERR_ITF_INCOMING_COMMAND_HAS_WRONG_VERSION + GVL_AdsInterface.wErrorIdOffset_IncomingAds; 			END_IF;
			
		IF iParTyp1 	<> PAR_TYPE_REGARDLESS 	THEN 
			IF localCmd.ParaCount1 	<> iParCount1 	THEN localRes.Error := GVL_AdsInterface_ERROR_IDS.ERR_ITF_INCOMING_COMMAND_HAS_WRONG_PARAMETER_COUNT + GVL_AdsInterface.wErrorIdOffset_IncomingAds; 	END_IF;
			IF localCmd.ParaTyp1	<> iParTyp1		THEN localRes.Error := GVL_AdsInterface_ERROR_IDS.ERR_ITF_INCOMING_COMMAND_HAS_WRONG_PARAMETER_TYP + GVL_AdsInterface.wErrorIdOffset_IncomingAds; 	END_IF;	
		END_IF;	
		
		IF iParTyp2 	<> PAR_TYPE_REGARDLESS THEN
			IF localCmd.ParaCount2 	<> iParCount2 	THEN localRes.Error := GVL_AdsInterface_ERROR_IDS.ERR_ITF_INCOMING_COMMAND_HAS_WRONG_PARAMETER_COUNT + GVL_AdsInterface.wErrorIdOffset_IncomingAds; 	END_IF;			
			IF localCmd.ParaTyp2	<> iParTyp2		THEN localRes.Error := GVL_AdsInterface_ERROR_IDS.ERR_ITF_INCOMING_COMMAND_HAS_WRONG_PARAMETER_TYP + GVL_AdsInterface.wErrorIdOffset_IncomingAds; 	END_IF;	
		END_IF
END_IF
END_METHOD

PROPERTY PUBLIC final P_EnabledInternally : bool
GET
P_EnabledInternally := bCmdEnabledByIntern;
END_GET
END_PROPERTY

END_FUNCTION_BLOCK

// Standard/Switch
{attribute 'hide'}
FUNCTION Switch : BOOL //Func to switch a boolean values. Returns the switched value
VAR_INPUT
	value : BOOL; //Original value to be switched
END_VAR

IF value THEN 
	value := FALSE;
ELSE 
	value := TRUE;
END_IF
Switch := value;

END_FUNCTION

// Logging/Logging
//Author: 				Walther Ronny
//Version:				1.4
//Last change:			07.02.18
//See Release notes at the bottom

PROGRAM Logging
VAR_OUTPUT
	WarningMsg : sErrorMsg;
	bWarning : BOOL;
END_VAR
VAR
	//ErrorMsg : sErrorMsg := (wComponent := USINT_TO_WORD(GVL.wCompId), sFunctionName := 'Logging');
//Msg buffer
	LogMsgBuf 			: ARRAY[0..(LOG_ARRAY_SIZE-1)] OF sLogMsgObject;	//Buffer to hold msg before written to a file
	iLoggingIdCounter 	: UDINT := 1;										//Counter to create unique Msg ID
	iCurBufIndex 		: UINT 	:= 0;										//Current buffer index to speed up inserting logs into buffer
	
//automatically updated variables	
	iCurFileSizeInKb 	: UINT;						//current size of log file (always updated)
	strCurSystemTime 	: STRING := EMPTY_STRING;	//current system time (always updated)
	strHostName			: STRING := 'NONE';			//name of target host
	
//help variables
	hDestFile 			: UINT;		//log file handle
	iErrId 				: UDINT;	//returning Beckhoff ADS error id. No use so far, just for debugging
	bDestTargetFound 	: BOOL;		//flag to tell if logging target pc/ beckhoff client is available

	pMsgObject 					: POINTER TO sLogMsgObject;	//retrieve log msg from buffer in order to write it to file when M_GetNextLogMsgtoWrite() is called
	bMsgReadyTobeLogged 		: BOOL;						//answers if there is a log msg to write to file when M_GetNextLogMsgtoWrite() is called
	bInitialTargetCheckDone,
	bTargetCheckDone			: BOOL;
	tTimerFileWriteIntervall 	: TON := (PT := Logging.LOG_FILE_WRITE_INTERVALL);
	
	LogPrgState 				: eLogPrgStates := eLogPrgStates.LOG_INITIALIZING;		//state machine variable
	
//Filepath variables	
	iFileNameNo  			: UINT 		:= 1; 				//Counter, if more than one log file per day is created
	strDestFileNameDate  	: STRING 	:= EMPTY_STRING; 	//Current date of log file	
    strDestFullPathName   	: STRING 	:= EMPTY_STRING;	//Full file path: directory + prefix + date + no + Ext
	
//File access Fb instances	 
	FileOpen 			: FB_FileOpen;			//Open/Create log file
	FilePuts 			: FB_FilePuts;			//Wirte strings to log file
	FileClose 			: FB_FileClose;			//Close log file
	FileRename	 		: FB_FileRename();
	FileDelete 			: FB_FileDelete();
	EnumFindFileEntry 	: FB_EnumFindFileEntry;	//TC_Utilities fb to get file size
	GetTime 			: NT_GetTime; 			//TC_Utilities fb to get system time
	GetHostName			: FB_GetHostName;		//TC_Utilities fb to get host name and check target access indirectly
	
//Configuration
	CurLogLevel 					: eLogLevel := eLogLevel.ALL; 	//Current loglevel. Note: ALL → TRACE → DEBUG → INFO → WARN → ERROR → FATAL → OFF.
	nCurLogBufferOccupancyInPct,
	iMaxLogBufferOccupancyInPct 	: UINT;	//Logs the maximum internal log buffer occupancy in percent since start-up, 100% means full
	iCurLogBufferOccupancy 			: UINT;	//Logs the current maximum internal log buffer occupancy in percent, 100% means full
	iMaxFileSizeInKB				: UINT := MAX_FILE_SIZE_IN_KB; //File size at which a new log file will be created. 50Mb max! 
	
	fTemp 							: LREAL;
	bInitializationByExternDone 	: BOOL;
END_VAR
VAR CONSTANT
	LOG_ARRAY_SIZE					: UINT			:= 1000;	//size of msg array	
	EMPTY_STRING 					: STRING 		:= '';
	MAX_FILE_SIZE_IN_KB 			: UINT 			:= 4096;	//File size at which a new log file will be created. 50Mb max! 
	LOG_FILE_WRITE_INTERVALL		: TIME			:= T#5S;	//intervall at which the log file is written - Note: Longer time => bigger Array
	TARGET_RECONNECT_TIME			: TIME			:= T#1M;	//if target not reachable, automatic reconnect try after that time
	FILE_ACCESS_FB_TIMEOUT			: TIME			:= T#3S;

	FILE_NAME_EXTENSION 			: STRING(4) 	:= '.txt'; 
END_VAR
VAR PERSISTENT
	strLastFileNameDate 	: STRING(10);	//holds the last filenamdate in order to decide whether use the same file or create a new one
	iLastFileNameCounter 	: UINT := 1;	//holds the last filenameno in order to decide whether use the same file or create a new one
END_VAR
(*
V1.0 Walther Ronny, 24.05.16
		- initial version
V1.1 Walther Ronny, 25.05.16
		- clean-up
		- P_LogLevel added
V1.2 Walther Ronny, 01.06.16
		- M_CheckTargetAccess
		- reconnect trys if target not availlable e.g. Pia Pc not started yet
V1.3 Walther Ronny, 28.08.17
		- eLogMode added (just two files instead keeping all)
V1.4 Werner Richter, 07.02.18
		- added configurable max file size with P_iMaxFileSizeKB
*)

//get actual system time from logging host target
	M_UpdateSysTimeVar();
	
//get current log file size
	M_UpdateCurFileSize();

//Execute write intervall timer
	tTimerFileWriteIntervall();

//set output variables
	WarningMsg.wComponent := GVL_Logging.wCompId;
	WarningMsg.ErrorTyp := eErrorTypes._WARNING;
	WarningMsg.sFunctionName := 'Logging';	

//state machine
CASE LogPrgState OF
//-----------------------------------------------------------------------------------------------------------------------
//Initial state which is called only once at FW start-up.  We need initial declaration of variables
//-----------------------------------------------------------------------------------------------------------------------
	eLogPrgStates.LOG_INITIALIZING : 
			
			IF strCurSystemTime <> EMPTY_STRING AND bInitializationByExternDone THEN
				
				//Update with persistent variable value
					iFileNameNo				:= iLastFileNameCounter;
					strDestFileNameDate 	:= strLastFileNameDate;
					
					LogPrgState := eLogPrgStates.LOG_STAND_BY;
			END_IF

//-----------------------------------------------------------------------------------------------------------------------
//Stand-by state which is called after writing was finished or Error. We are waiting for 
//a) write intervall timer or 
//b) host availability or 
//c) log messages to arrive
//-----------------------------------------------------------------------------------------------------------------------			
	eLogPrgStates.LOG_STAND_BY:	//Waiting for log interval timer to finish

										
			tTimerFileWriteIntervall.IN := TRUE;
			
			IF tTimerFileWriteIntervall.Q THEN
				tTimerFileWriteIntervall.IN := FALSE;
				
				M_CheckTargetAccess(bDone => bTargetCheckDone);
				
				IF bTargetCheckDone THEN
					bInitialTargetCheckDone := TRUE;
				END_IF
				
				IF bDestTargetFound AND bInitialTargetCheckDone THEN
					bWarning := FALSE;
	
					M_UpdateFilePath();
					
					M_GetNextLogMsgtoWrite(	bNextMsgAvailable 	=> bMsgReadyTobeLogged,
											pMsgObject 			=> );
											
					IF bMsgReadyTobeLogged THEN				
						LogPrgState := eLogPrgStates.LOG_OPENING_FILE;				
						
					END_IF
				ELSIF bTargetCheckDone THEN			
					bDestTargetFound := FALSE;
						
					WarningMsg.wErrorNo := GVL_Logging_ERROR_IDS.ERR_LOG_FILE_TARGET_NOT_FOUND + GVL_Logging.wErrorIdOffset;	
					bWarning := TRUE;
					ErrorManagement.M_InsertNewError(ErrorMsg := WarningMsg);						
				ELSE
					;
					//nothing, we wait until target chack is finished
				END_IF
				
			END_IF

//-----------------------------------------------------------------------------------------------------------------------
//opening/creating log file and get handle
//-----------------------------------------------------------------------------------------------------------------------		
	eLogPrgStates.LOG_OPENING_FILE :
				
			FileOpen(	bExecute	:= TRUE,
						sNetId 		:= GVL_Logging.DEST_AMS_NET_ID,
						sPathName 	:= strDestFullPathName,
						ePath		:= PATH_GENERIC,
						nMode 		:= FOPEN_MODEAPPEND OR FOPEN_MODETEXT,
						tTimeout 	:= FILE_ACCESS_FB_TIMEOUT,
						bError 		=> ,
						nErrId		=> iErrId,
						hFile 		=> hDestFile );
						
			IF NOT FileOpen.bBusy THEN
				IF FileOpen.bError THEN
					
					WarningMsg.wErrorNo := GVL_Logging_ERROR_IDS.ERR_LOG_FILE_COULD_NOT_BE_OPENED_OR_CREATED + GVL_Logging.wErrorIdOffset;
					bWarning := TRUE;
					ErrorManagement.M_InsertNewError(ErrorMsg := WarningMsg);	
					
					logPrgState := eLogPrgStates.LOG_ERROR;					
					
				ELSE
					bWarning := FALSE;
					LogPrgState := eLogPrgStates.LOG_WRITING_FILE;
					
				END_IF
				//Reset fb
					FileOpen(bExecute := FALSE);
					
			END_IF
			
//-----------------------------------------------------------------------------------------------------------------------
//writing log file with data from the internal logging buffer - Line after Line until no message left
//-----------------------------------------------------------------------------------------------------------------------			
	eLogPrgStates.LOG_WRITING_FILE:
				M_GetNextLogMsgtoWrite(	bNextMsgAvailable 	=> bMsgReadyTobeLogged,
										pMsgObject 			=> pMsgObject);
				
				IF bMsgReadyTobeLogged THEN
					FilePuts(	sNetId		:= GVL_Logging.DEST_AMS_NET_ID, 
								hFile		:= hDestFile,
								sLine 		:= M_CreateLogString(pMsgObject),                  
								bExecute	:= TRUE, 
								tTimeout	:= FILE_ACCESS_FB_TIMEOUT);
						
					IF NOT FilePuts.bBusy THEN //Done
						IF FilePuts.bError THEN
							WarningMsg.wErrorNo := GVL_Logging_ERROR_IDS.ERR_STRING_COULD_NOT_BE_WRITTEN_TO_THE_OPENED_LOG_FILE + GVL_Logging.wErrorIdOffset;
							bWarning := TRUE;
							ErrorManagement.M_InsertNewError(ErrorMsg := WarningMsg);	
							
							LogPrgState := eLogPrgStates.LOG_ERROR;
							
						ELSE
							bWarning := FALSE;
							
							//delete msg, thus it was sent
								pMsgObject^.bIsValidMsg := FALSE;
								
							Dec(iCurLogBufferOccupancy);	
						END_IF
						
						FilePuts(bExecute:= FALSE);
					END_IF	
				
				ELSE //No more msg to write, thus let´s close the file
						LogPrgState := eLogPrgStates.LOG_CLOSING_FILE;
					
				END_IF
//-----------------------------------------------------------------------------------------------------------------------
// closing log file and returning to stand-by
//-----------------------------------------------------------------------------------------------------------------------			
	eLogPrgStates.LOG_CLOSING_FILE: //Close file 

				FileClose(	bExecute	:= TRUE,
							sNetId 		:= GVL_Logging.DEST_AMS_NET_ID,
							tTimeout 	:= FILE_ACCESS_FB_TIMEOUT,
							bError 		=> ,
							hFile 		:= hDestFile );
							
				IF NOT FileClose.bBusy THEN
					IF FileClose.bError THEN
						WarningMsg.wErrorNo := GVL_Logging_ERROR_IDS.ERR_LOG_FILE_COULD_NOT_BE_CLOSED + GVL_Logging.wErrorIdOffset;					
						bWarning := TRUE;
						ErrorManagement.M_InsertNewError(ErrorMsg := WarningMsg);	
						
						LogPrgState := eLogPrgStates.LOG_ERROR;
						
					ELSE
						bWarning := FALSE;
						LogPrgState := eLogPrgStates.LOG_STAND_BY;
	
					END_IF	
					FileClose(bExecute := FALSE);				
				END_IF
				
//-----------------------------------------------------------------------------------------------------------------------
//Error opening/creating/closing a log file. Implicit transition to stand-by state
//-----------------------------------------------------------------------------------------------------------------------	
	eLogPrgStates.LOG_ERROR : 
				//try again
					LogPrgState := eLogPrgStates.LOG_STAND_BY;
END_CASE

//Update occupancy counter
fTemp := (100 * iCurLogBufferOccupancy) / TO_LREAL(LOG_ARRAY_SIZE);	
nCurLogBufferOccupancyInPct := TO_UINT(fTemp);				
IF  nCurLogBufferOccupancyInPct > iMaxLogBufferOccupancyInPct THEN
	iMaxLogBufferOccupancyInPct := nCurLogBufferOccupancyInPct;						
END_IF

METHOD PUBLIC Debug
VAR_INPUT
	Caller 	: STRING;
	Msg 	: STRING(255);
END_VAR
VAR
	LogMsg : sLogMsg;
END_VAR
LogMsg.LogLevel 			:= eLogLevel.DEBUG;
LogMsg.sCallFunctionName 	:= Caller;
LogMsg.sLogMessage 			:= Msg;

M_InsertLog(LogMsg := LogMsg);
END_METHOD

METHOD PUBLIC Error
VAR_INPUT
	Caller 	: STRING;
	Msg 	: STRING(255);
END_VAR
VAR
	LogMsg : sLogMsg;
END_VAR
LogMsg.LogLevel 			:= eLogLevel.ERROR;
LogMsg.sCallFunctionName 	:= Caller;
LogMsg.sLogMessage 			:= Msg;

M_InsertLog(LogMsg := LogMsg);
END_METHOD

METHOD PUBLIC Fatal
VAR_INPUT
	Caller 	: STRING;
	Msg 	: STRING(255);
END_VAR
VAR
	LogMsg : sLogMsg;
END_VAR
LogMsg.LogLevel 			:= eLogLevel.FATAL;
LogMsg.sCallFunctionName 	:= Caller;
LogMsg.sLogMessage 			:= Msg;

M_InsertLog(LogMsg := LogMsg);
END_METHOD

METHOD PUBLIC Info
VAR_INPUT
	Caller 	: STRING;
	Msg 	: STRING(255);
END_VAR
VAR
	LogMsg : sLogMsg;
END_VAR
LogMsg.LogLevel 			:= eLogLevel.INFO;
LogMsg.sCallFunctionName 	:= Caller;
LogMsg.sLogMessage 			:= Msg;

M_InsertLog(LogMsg := LogMsg);
END_METHOD

METHOD PUBLIC M_Initialize
VAR_INPUT
	wCompId 			: tErrorConstant;		//TRUE => Logging activated, FALSE => Logging deactivated
	wErrorIdOffset		: tErrorConstant;		//Offset to be added to all ErrorId´s
	TDesAmsNetId 		: T_AmsNetId; 		
	sFileDestinationDir : STRING;
	sFileNamePrefix  	: STRING(20); 
	eLogMode 			: E_LogModes;
END_VAR
IF  bInitializationByExternDone THEN
	RETURN;
END_IF

GVL_Logging.wCompId 					:= wCompId;
GVL_Logging.wErrorIdOffset 				:= wErrorIdOffset;

GVL_Logging.DEST_AMS_NET_ID 			:= TDesAmsNetId;
GVL_Logging.FILE_DESTINATION_DIRECTORY 	:= sFileDestinationDir;
GVL_Logging.FILE_NAME_PREFIX 			:= sFileNamePrefix;
GVL_Logging.eLogMode 					:= eLogMode;

bInitializationByExternDone := TRUE;
END_METHOD

PROPERTY PUBLIC P_bAllDataWritten : bool
GET
	M_GetNextLogMsgtoWrite(	bNextMsgAvailable 	=> bMsgReadyTobeLogged,
							pMsgObject 			=> );
				
	IF NOT bMsgReadyTobeLogged AND 	LogPrgState = eLogPrgStates.LOG_STAND_BY THEN
		P_bAllDataWritten := TRUE;
	ELSE
		P_bAllDataWritten := FALSE;

	END_IF
END_GET
END_PROPERTY

PROPERTY public P_bResetMaxLogBufferOccupancyInPct : BOOL
SET
IF P_bResetMaxLogBufferOccupancyInPct THEN
	iMaxLogBufferOccupancyInPct := 0;
END_IF
END_SET
END_PROPERTY

PROPERTY public P_iMaxFileSizeKB : UINT
GET
P_iMaxFileSizeKB := iMaxFileSizeInKB;
END_GET
SET
iMaxFileSizeInKB := P_iMaxFileSizeKB;
END_SET
END_PROPERTY

PROPERTY PUBLIC P_iMaxLogBufferOccupancyInPct : uint
GET
P_iMaxLogBufferOccupancyInPct := iMaxLogBufferOccupancyInPct;
END_GET
END_PROPERTY

PROPERTY PUBLIC P_LogLevel : eLogLevel
GET
P_LogLevel := CurLogLevel;
END_GET
SET
CurLogLevel := P_LogLevel;
END_SET
END_PROPERTY

PROPERTY PUBLIC P_LogPrgState :  eLogPrgStates
GET
P_LogPrgState := LogPrgState;
END_GET
END_PROPERTY

PROPERTY PUBLIC P_nCurLogBufferOccupancyInPct : uint
GET
P_nCurLogBufferOccupancyInPct := nCurLogBufferOccupancyInPct;
END_GET
END_PROPERTY

METHOD PUBLIC Trace
VAR_INPUT
	Caller 	: STRING;
	Msg 	: STRING(255);
END_VAR
VAR
	LogMsg : sLogMsg;
END_VAR
LogMsg.LogLevel 			:= eLogLevel.TRACE;
LogMsg.sCallFunctionName 	:= Caller;
LogMsg.sLogMessage 			:= Msg;

M_InsertLog(LogMsg := LogMsg);
END_METHOD

METHOD PUBLIC Warn
VAR_INPUT
	Caller 	: STRING;
	Msg 	: STRING(255);
END_VAR
VAR
	LogMsg : sLogMsg;
END_VAR
LogMsg.LogLevel 			:= eLogLevel.WARN;
LogMsg.sCallFunctionName 	:= Caller;
LogMsg.sLogMessage 			:= Msg;

M_InsertLog(LogMsg := LogMsg);
END_METHOD

{attribute 'hide'}
METHOD PRIVATE M_CheckTargetAccess
VAR_OUTPUT
	bDone : BOOL;
END_VAR
VAR	
	strHostName_tmp : STRING;
END_VAR

GetHostName(sNetID 		:= GVL_Logging.DEST_AMS_NET_ID,
			tTimeout 	:= T#500MS,
			bExecute 	:= TRUE,
			sHostName 	=> strHostName_tmp);
		
IF NOT GetHostName.bBusy THEN
	IF GetHostName.bError THEN
		bDestTargetFound 	:= FALSE;
		strHostName 		:= 'NONE';
		
	ELSE
		bDestTargetFound 	:= TRUE;
		strHostName 		:= strHostName_tmp ;	
		
	END_IF
		bDone := TRUE;
		
	//Reset
		GetHostName(bExecute := FALSE);
END_IF
END_METHOD

{attribute 'hide'}
METHOD PRIVATE M_CreateLogString : string(255)
VAR_INPUT
	pMsgObject : POINTER TO sLogMsgObject;
END_VAR
VAR 
	strLogLevel : STRING;
	strLog : STRING(255);
END_VAR
//Timestamp
	strLog := concat('[',pMsgObject^.sTimeStamp);
	strLog := concat(strLog,'] ');

//Loglevel
	CASE pMsgObject^.LogMsg.LogLevel OF
		eLogLevel.WARN 	:	strLogLevel := 'WARN ';
		eLogLevel.INFO 	:	strLogLevel := 'INFO ';
		eLogLevel.ERROR :	strLogLevel := 'ERROR';
		eLogLevel.DEBUG :	strLogLevel := 'DEBUG';
		eLogLevel.TRACE :	strLogLevel := 'TRACE';
		eLogLevel.FATAL :	strLogLevel := 'FATAL';
	END_CASE
	
	strLog := CONCAT(strLog, strLogLevel);
	strLog := CONCAT(strLog, ' ');

//Log message
	strLog := CONCAT(strLog, pMsgObject^.LogMsg.sCallFunctionName);
	strLog := CONCAT(strLog, ' - ');
	strLog := CONCAT(strLog, pMsgObject^.LogMsg.sLogMessage);

//string end
	strLog := CONCAT(strLog, '');
	strLog := CONCAT(strLog, '$L');

//Pass final string	
	M_CreateLogString := strLog;
END_METHOD

{attribute 'hide'}
METHOD PRIVATE M_DeleteFile : T_RETVALUE //no error message sent if failed!
VAR_INPUT
	strFilepath : STRING;
END_VAR
VAR
	eRetVal : T_RETVALUE;
END_VAR
FileDelete(	sNetId 		:= GVL_Logging.DEST_AMS_NET_ID,
			sPathName 	:= strFilepath,
			bExecute 	:= TRUE, 
			tTimeout 	:= FILE_ACCESS_FB_TIMEOUT,
			ePath 		:= PATH_GENERIC
			);
IF NOT FileDelete.bBusy THEN
	eRetVal := eOK;
	FileDelete(bExecute := FALSE);
END_IF

M_DeleteFile := eRetVal;
END_METHOD

{attribute 'hide'}
METHOD PRIVATE M_GenerateFilepath : STRING
VAR_INPUT
	strDirectory  		: STRING; 
	strFileNamePref  	: STRING; 
	strFileNameDate  	: STRING(10); 
	iFileNameNo  		: UINT; 
	strFileNameInfo		: STRING(5);
	strFileNameExt		: STRING(4);
END_VAR
VAR	
	filepath : STRING;  
END_VAR
IF GVL_Logging.eLogMode = E_LogModes.KeepAllFiles THEN
	filepath := CONCAT(strDirectory, strFileNamePref);
	filepath := CONCAT(filepath, '_');
	filepath := CONCAT(filepath, strFileNameDate);
	filepath := CONCAT(filepath, '_');
	filepath := CONCAT(filepath, UINT_TO_STRING(iFileNameNo));
	filepath := CONCAT(filepath, strFileNameInfo);
	filepath := CONCAT(filepath, strFileNameExt);
	
ELSIF GVL_Logging.eLogMode = E_LogModes.KeepTwoFiles THEN
	filepath := CONCAT(strDirectory, strFileNamePref);
	IF strFileNameInfo <> '' THEN
		filepath := CONCAT(filepath, '_');
	END_IF
	filepath := CONCAT(filepath, strFileNameInfo);
	filepath := CONCAT(filepath, strFileNameExt);
	
END_IF
M_GenerateFilepath := filepath;
END_METHOD

{attribute 'hide'}
METHOD PRIVATE M_GetNextLogMsgtoWrite
VAR_OUTPUT
	bNextMsgAvailable : BOOL;
	pMsgObject : POINTER TO sLogMsgObject;
END_VAR
VAR
	i : UINT;
	iSmallestId : UDINT := 16#FFFFFFFF;
END_VAR
//find oldest message => smalled id
	FOR i := 0 TO (LOG_ARRAY_SIZE - 1) DO		
		IF LogMsgBuf[i].bIsValidMsg THEN //0 => empty
			
			IF LogMsgBuf[i].iLogMsgId < iSmallestId THEN
				iSmallestId := LogMsgBuf[i].iLogMsgId;
				
				bNextMsgAvailable := TRUE;
				pMsgObject := ADR(LogMsgBuf[i]);
			END_IF
		END_IF
	END_FOR
END_METHOD

{attribute 'hide'}
METHOD public M_InsertLog
VAR_INPUT
	LogMsg : sLogMsg;
END_VAR
VAR
	i : UINT;
END_VAR
IF LogMsg.LogLevel <= CurLogLevel THEN

		IF iCurBufIndex >= LOG_ARRAY_SIZE - 1 THEN
			iCurBufIndex := 0;
			
		END_IF
	
		FOR i := iCurBufIndex TO (LOG_ARRAY_SIZE - 1) DO
			
			IF NOT LogMsgBuf[iCurBufIndex].bIsValidMsg THEN //0 => empty
				
				LogMsgBuf[iCurBufIndex].bIsValidMsg	:= TRUE;
				LogMsgBuf[iCurBufIndex].iLogMsgId 	:= iLoggingIdCounter;
				LogMsgBuf[iCurBufIndex].LogMsg 		:= LogMsg;
				LogMsgBuf[iCurBufIndex].sTimeStamp	:= strCurSystemTime;
				
				Inc(iCurBufIndex);
				iLoggingIdCounter := iLoggingIdCounter + 1;
				
				Inc(iCurLogBufferOccupancy);
				
				bMsgReadyTobeLogged := TRUE;
				EXIT;
				
			END_IF
		END_FOR
END_IF
END_METHOD

{attribute 'hide'}
METHOD PRIVATE M_RenameFile : T_RETVALUE
VAR_INPUT
	strNewFilepath : STRING;
END_VAR
VAR
	eRetVal : T_RETVALUE;
END_VAR
FileRename(	sNetId 		:= GVL_Logging.DEST_AMS_NET_ID,
			sNewName 	:= strNewFilepath,
			sOldName 	:= strDestFullPathName, 
			bExecute 	:= TRUE, 
			tTimeout 	:= FILE_ACCESS_FB_TIMEOUT,
			ePath 		:= PATH_GENERIC
			);
IF NOT FileRename.bBusy THEN
	eRetVal := eBUSY;
	IF FileRename.bError THEN
		eRetVal := eNOK;
		WarningMsg.wErrorNo := GVL_Logging_ERROR_IDS.ERR_STRING_COULD_NOT_BE_WRITTEN_TO_THE_OPENED_LOG_FILE + GVL_Logging.wErrorIdOffset;
		bWarning := TRUE;
		ErrorManagement.M_InsertNewError(ErrorMsg := WarningMsg);
		LogPrgState := eLogPrgStates.LOG_ERROR;	
	ELSE
		eRetVal := eOK;
	END_IF	
	FileRename(bExecute := FALSE);
END_IF

M_RenameFile := eRetVal;
END_METHOD

{attribute 'hide'}
METHOD PRIVATE M_UpdateCurFileSize
VAR
	fileinfo 	: ST_FindFileEntry;
	maxSize 	: DWORD;
	//curSize : DWORD;
END_VAR

EnumFindFileEntry(	sNetID 		:= GVL_Logging.DEST_AMS_NET_ID, 
					tTimeout 	:= FILE_ACCESS_FB_TIMEOUT, 
					sPathName 	:= strDestFullPathName,
					bExecute 	:= TRUE,
					stFindFile	=> fileinfo );
					
IF NOT EnumFindFileEntry.bBusy THEN
	
	IF EnumFindFileEntry.bError THEN
		iCurFileSizeInKb := 0;
	
	ELSE		
		iCurFileSizeInkb := DWORD_TO_UINT(SHR(fileinfo.fileSize.dwLowPart,10));
					
	END_IF
	
	EnumFindFileEntry(bExecute := FALSE);
END_IF
END_METHOD

{attribute 'hide'}
METHOD PRIVATE M_UpdateFilePath
VAR
	strHlpString : STRING;
	strCurDate 	: STRING(10)	:= LEFT(strCurSystemTime, 10); 			//get only yyyy-mm-dd
END_VAR
IF GVL_Logging.eLogMode = E_LogModes.KeepAllFiles THEN
	//Check current conditions
		IF strCurDate <> strLastFileNameDate THEN			//date changed		
			//Reset counter					
				iFileNameNo := 1;			
			//Set new date
				strDestFileNameDate := strCurDate;
				
		ELSIF iCurFileSizeInKb >= iMaxFileSizeInKB THEN	//file size exceeded			
			//inc counter
				Inc(iFileNameNo);

		ELSE
			//nothing to do here

		END_IF
		
	//Update full file path	
		strDestFullPathName :=	M_GenerateFilepath(	strDirectory 	:= GVL_Logging.FILE_DESTINATION_DIRECTORY,
													strFileNamePref := GVL_Logging.FILE_NAME_PREFIX,
													strFileNameDate := strDestFileNameDate,
													iFileNameNo 	:= iFileNameNo,
													strFileNameInfo := '',
													strFileNameExt 	:= FILE_NAME_EXTENSION);

//Update persistent variables
	iLastFileNameCounter 	:= iFileNameNo;
	strLastFileNameDate		:= strDestFileNameDate;
	
ELSIF GVL_Logging.eLogMode = E_LogModes.KeepTwoFiles THEN
	//Update full file path	
		strDestFullPathName :=	M_GenerateFilepath(	strDirectory 	:= GVL_Logging.FILE_DESTINATION_DIRECTORY,
													strFileNamePref := GVL_Logging.FILE_NAME_PREFIX,
													strFileNameDate := '',
													iFileNameNo 	:= 1,
													strFileNameInfo := '',
													strFileNameExt 	:= FILE_NAME_EXTENSION);

	IF iCurFileSizeInKb >= iMaxFileSizeInKB THEN	//file size exceeded	
		strHlpString := M_GenerateFilepath(	strDirectory 	:= GVL_Logging.FILE_DESTINATION_DIRECTORY,
												strFileNamePref := GVL_Logging.FILE_NAME_PREFIX,
												strFileNameDate := '',
												iFileNameNo 	:= 0,
												strFileNameInfo := GVL_Logging.FILE_NAME_EXT_OLD,
												strFileNameExt 	:= FILE_NAME_EXTENSION
												);
		
		M_DeleteFile(strHlpString);	//if a "old" file exists already, we delete it
		M_RenameFile(strHlpString); //current file gets renamed marked "old"	
		iCurFileSizeInKb := 0;
	END_IF
end_if
END_METHOD

{attribute 'hide'}
METHOD PRIVATE M_UpdateSysTimeVar
VAR	
	curTimeStruct : TIMESTRUCT;
END_VAR

GetTime(NETID := GVL_Logging.DEST_AMS_NET_ID, //get local time
		TMOUT := t#500ms,
		START := TRUE,
		TIMESTR => curTimeStruct);
		
IF NOT GetTime.BUSY THEN
	IF GetTime.ERR THEN
		strCurSystemTime := 'Error while generating timestamp';
	
	ELSE
		strCurSystemTime := SYSTEMTIME_TO_STRING(curTimeStruct);		
	END_IF
	
	//Reset
		GetTime(START := FALSE);
END_IF
END_METHOD

END_PROGRAM

// ErrorManagement/ErrorManagement
//Author: 				Koster Daniel, Walther Ronny
//Version:				1.70
//Last change:			25.10.2019
//See Release notes at the bottom
//{attribute 'hide_all_locals'}
PROGRAM ErrorManagement
VAR
	pErrHnd : POINTER TO FB_ErrorHandler_Base;
	
	iSysErrorMsgIdCounter :		UINT := 1;		//Counter to create unique ErrorMsg ID
	SysErrorList:				ARRAY[0..(ERROR_ARRAY_SIZE-1)] OF sSystemError;
	

	//Automatic periodical Event sending
		tEventIntervalTime : 		TIME := ERROR_EVENT_SENDING_CYCLE_TIME;
		tEventIntervalTimer :		TON;
		iEvtSendingIndex :			UINT := 0;	//Index while scrolling thru error list inside M_SendEvents method
	
	//Event sending mode flags	
		CurNotificationMode : 			eErrorNotificationMode := ERROR_NOTIFICATION_MODE;
		
		bEventSendingOnceActive : 		BOOL := FALSE;	

//Note: The following objects are used like constants, but thus wComponent is set first when the program is initialized they can not be declared as constants!
	NULL_ERROR_MSG : 	sErrorMsg 		:= (	wModule 		:= 1,
												pErrorHandler 	:= ADR(ErrHand_Dummy),
												wComponent 		:= GVL_ErrorManagement.wCompId,
												sFunctionName 	:= '***NULL_ERROR***',
												ErrorTyp		:= eErrorTypes._ERROR,
												wErrorNo 		:= GVL.ERR_NO_ERROR);	
	
	NULL_ERROR : 		sSystemError 	:= (	SysErrorMessageID 	:= 0,
												ErrorMsg 			:= NULL_ERROR_MSG);	
	ErrHand_Dummy :		FB_ErrorHandler_Base;												
END_VAR
VAR CONSTANT
	ERROR_ARRAY_SIZE:					UINT:= 40;			//size of error array
	ERROR_NOTIFICATION_MODE :			UINT := eErrorNotificationMode.SENDING_ERRORS_ONCE_IMMEDIATLY;
	ERROR_EVENT_SENDING_CYCLE_TIME : 	TIME := T#200MS;	//periodic event sending intervall
	

								
	EMPTY_SYS_ERROR : 	sSystemError 	:= (	SysErrorMessageID 	:= 0);	
	

END_VAR
(*
V1.0 Koster Daniel
		- initial version
V1.1 Walther Ronny, 26.01.16 complete rework:
		- automatic msg id
		- 3 sending modes included
		- sSystemError struct changed
		- sSystemErrorEvent changed
		- Errorhandler option included 
V1.2 Walther Ronny, 19.02.16 minor change:
		-  sending "Null-Error" event included inside M_RemoveAllErrors 
V1.3 Walther Ronny, 22.02.16 minor change
		-  bool return value from methods removed
V1.4 Walther Ronny, 16.03.16 minor change
		-  Bugfix: sending immediatly => keep min cycle time when sending many errors
V1.5 Walther Ronny, 19.05.16 minor change		
		- P_bHaveAllErrorsBeenSentAtLeastOnce included
V1.6 Walther Ronny, 23.05.16 minor change		
		- forwarding to Logging.prg included
		- EMPTY_SYS_ERROR and NULL_ERROR constant added
V1.70 Werner Richter, 25.10.2019
		- M_SendEvents, delete error after sending, if it is a warning to preven array overflow
		- M_InsertNewError, if counter is 0xffff reset it and remove all errors
*)

//automatic sending modes
	M_SendEvents();

METHOD PUBLIC M_GetErrorArrayInformation
VAR_OUTPUT
	iErrorCount,
	iFreeSpaceCount :		UINT := 0;	
	
	bMethodError : 			BOOL := FALSE;
	MethodErrorMsg : 		sErrorMsg;
END_VAR
VAR
	i : UINT;
END_VAR
(*
V1.0  Walther Ronny, 27.12.15
		- initial version
*)
MethodErrorMsg.wComponent 		:= GVL_ErrorManagement.wCompId;
MethodErrorMsg.sFunctionName 	:= 'M_GetErrorArrayInformation';
MethodErrorMsg.wErrorNo 		:= GVL.ERR_NO_ERROR;

//scroll errors
	 FOR i := 0 TO (ERROR_ARRAY_SIZE - 1) DO
		
		IF SysErrorList[i].SysErrorMessageID = 0 THEN //0 => empty THEN
			//Determine free spaces
		 		inc(iFreeSpaceCount);
			
		ELSE
			//Count errors
				inc(iErrorCount);
				
		END_IF								
	END_FOR
END_METHOD

METHOD PUBLIC M_GetErrorInfo : sSystemError	//Gives back the Info for the SysError with ErrorID = ErrorID
VAR_INPUT
	iSysErrorMsgId:	UINT;
END_VAR
VAR_OUTPUT
	bErrorMsgIdFound : 	BOOL := FALSE;
	bMethodError : 		BOOL := FALSE;
	MethodErrorMsg : 	sErrorMsg;
END_VAR
VAR 
	i : UINT;
END_VAR
MethodErrorMsg.wComponent 		:= GVL_ErrorManagement.wCompId;
MethodErrorMsg.sFunctionName 	:= 'M_GetErrorInfo';
MethodErrorMsg.wErrorNo 		:= GVL.ERR_NO_ERROR;

IF iSysErrorMsgId = 0 THEN		
	bMethodError := TRUE;
	MethodErrorMsg.wErrorNo := GVL_ErrorManagement_ERROR_IDS.ERR_ERROR_ID_ZERO_INVALID + GVL_ErrorManagement.wErrorIdOffset;
	
ELSE
	FOR i := 0 TO (ERROR_ARRAY_SIZE - 1) DO
		IF SysErrorList[i].SysErrorMessageID = iSysErrorMsgId THEN	//ErrorID is found
			bErrorMsgIdFound := TRUE;			
			
			M_GetErrorInfo := SysErrorList[i];
			EXIT;			
		END_IF
	END_FOR
END_IF

IF NOT bErrorMsgIdFound THEN//If ErrorID couldn´t be found
	bMethodError := TRUE;
	MethodErrorMsg.wErrorNo := GVL_ErrorManagement_ERROR_IDS.ERR_ERROR_ID_NOT_FOUND + GVL_ErrorManagement.wErrorIdOffset;
	
END_IF
END_METHOD

METHOD PUBLIC M_Initialize
VAR_INPUT
	wCompId 		: tErrorConstant;	//TRUE => Logging activated, FALSE => Logging deactivated
	wErrorIdOffset	: tErrorConstant;	//Offset to be added to all ErrorId´s	
	bLoggingOnOff 	: BOOL;				//TRUE => Logging activated, FALSE => Logging deactivated
	pEvt 			: POINTER TO sSystemErrorEvent;
END_VAR
GVL_ErrorManagement.wCompId 		:= wCompId;
GVL_ErrorManagement.wErrorIdOffset 	:= wErrorIdOffset;
GVL_ErrorManagement.bLoggingOnOff	:= bLoggingOnOff;


//Check Evt pointer, if invalid set dummy
	IF IsValidPtr(pEvt) THEN
		GVL_ErrorManagement.pEvt 			:= pEvt;
		
	ELSE		
		GVL_ErrorManagement.pEvt := ADR(GVL_ErrorManagement.cDUMMY_EVENT);

	END_IF
END_METHOD

METHOD PUBLIC M_InsertNewError		//Puts new SysError in the SysError List
VAR_INPUT
		ErrorMsg 		: sErrorMsg;
END_VAR
VAR_OUTPUT
	iSysErrorMsgId : 	UINT := 0;
	bMethodError : 		BOOL := FALSE;
	MethodErrorMsg : 	sErrorMsg;
END_VAR
VAR
	bErrorSet : 		BOOL := FALSE;
	i : 				UINT := 0;
END_VAR
MethodErrorMsg.wComponent 		:= GVL_ErrorManagement.wCompId;
MethodErrorMsg.sFunctionName 	:= 'M_InsertNewSysError';
MethodErrorMsg.wErrorNo 		:= GVL.ERR_NO_ERROR;


FOR i := 0 TO (ERROR_ARRAY_SIZE - 1) DO
	IF SysErrorList[i].SysErrorMessageID = 0 THEN //0 => empty
		iSysErrorMsgId := iSysErrorMsgIdCounter;
		
		SysErrorList[i].SysErrorMessageID 	:= iSysErrorMsgId;
		SysErrorList[i].ErrorMsg 			:= ErrorMsg;	
		SysErrorList[i].bErrorWasSent		:= FALSE;
		
		//Handle not set variables
			IF NOT IsValidPtr(SysErrorList[i].ErrorMsg.pErrorHandler) THEN
				SysErrorList[i].ErrorMsg.pErrorHandler := ADR(ErrHand_Dummy);
			END_IF
			IF SysErrorList[i].ErrorMsg.ErrorTyp = eErrorTypes._UNDEFINED THEN //otherwise 0 is always a fatal error for PIA
				 SysErrorList[i].ErrorMsg.ErrorTyp := eErrorTypes._ERROR;
			END_IF
		//Logging
			M_CreateLogData(pErr := SysErrorList[i]);
			
		// reset if too much warnings were sent	
		IF iSysErrorMsgIdCounter >= 16#FFFF THEN
			iSysErrorMsgIdCounter := 0;
			M_RemoveAllErrors();		
		END_IF
	
		inc(iSysErrorMsgIdCounter);
		bErrorSet := TRUE;
		
		EXIT;
	END_IF
END_FOR

IF NOT bErrorSet THEN
	MethodErrorMsg.wErrorNo 		:= GVL_ErrorManagement_ERROR_IDS.ERR_ERROR_ARRAY_FULL + GVL_ErrorManagement.wErrorIdOffset;
	bMethodError := TRUE;
END_IF
END_METHOD

METHOD PUBLIC M_RemoveAllErrors
VAR_OUTPUT
	bMethodError : 		BOOL := FALSE;
	MethodErrorMsg : 	sErrorMsg;
END_VAR
VAR
	i : UINT;
	sysErr : sSystemError;
END_VAR
MethodErrorMsg.wComponent 		:= GVL_ErrorManagement.wCompId;
MethodErrorMsg.sFunctionName 	:= 'M_RemoveAllErrors';
MethodErrorMsg.wErrorNo 		:= GVL.ERR_NO_ERROR;


sysErr := NULL_ERROR;
sysErr.ErrorMsg.wComponent := GVL_ErrorManagement.wCompId;

FOR i := 0 TO (ERROR_ARRAY_SIZE - 1) DO
	SysErrorList[i] := EMPTY_SYS_ERROR;
END_FOR

//Log data	
	M_CreateLogData(pErr := sysErr);

//Create Event - NULL ERROR	
	M_CreateEvent(sysErr := sysErr);
END_METHOD

METHOD public M_RemoveError	//Clears SysError with ErrorID = ErrorID
VAR_INPUT
	iSysErrorMsgId : 	UINT;
END_VAR
VAR_OUTPUT
	bErrorMsgIdFound : 	BOOL := FALSE;
	bMethodError : 		BOOL := FALSE;
	MethodErrorMsg : 	sErrorMsg;
END_VAR
VAR
	i : UINT;
END_VAR
MethodErrorMsg.wComponent 		:= GVL_ErrorManagement.wCompId;
MethodErrorMsg.sFunctionName 	:= 'M_RemoveError';
MethodErrorMsg.wErrorNo 		:= GVL.ERR_NO_ERROR;

IF iSysErrorMsgId = 0 THEN		
	bMethodError := TRUE;
	MethodErrorMsg.wErrorNo := GVL_ErrorManagement_ERROR_IDS.ERR_ERROR_ID_ZERO_INVALID + GVL_ErrorManagement.wErrorIdOffset;
	
ELSE
	FOR i := 0 TO (ERROR_ARRAY_SIZE - 1) DO
		IF SysErrorList[i].SysErrorMessageID = iSysErrorMsgId THEN	//ErrorID is found
			bErrorMsgIdFound := TRUE;			
			
			SysErrorList[i] := EMPTY_SYS_ERROR;	//remove SysError
			EXIT;			
		END_IF
	END_FOR
END_IF

IF NOT bErrorMsgIdFound THEN//If ErrorID couldn´t be found
	bMethodError := TRUE;
	MethodErrorMsg.wErrorNo := GVL_ErrorManagement_ERROR_IDS.ERR_ERROR_ID_NOT_FOUND + GVL_ErrorManagement.wErrorIdOffset;
	
END_IF
END_METHOD

METHOD PUBLIC M_ResetSysErrorMng
M_RemoveAllErrors();
END_METHOD

METHOD PUBLIC M_SendAllErrorOnce
VAR_OUTPUT
	bMethodError : 		BOOL := FALSE;
	MethodErrorMsg : 	sErrorMsg;
END_VAR
MethodErrorMsg.wComponent 		:= GVL_ErrorManagement.wCompId;
MethodErrorMsg.sFunctionName 	:= 'M_SendEvtOnce';
MethodErrorMsg.wErrorNo 		:= GVL.ERR_NO_ERROR;

IF CurNotificationMode = eErrorNotificationMode.SENDING_ERRORS_ALWAYS_PERIODICALLY THEN
	bMethodError := TRUE;
	MethodErrorMsg.wErrorNo 	:= GVL_ErrorManagement_ERROR_IDS.ERR_SEND_ERRORS_ONCE_NOT_POSSIBLE_THUS_PERIODIC_SENDING_ACTIVATED + GVL_ErrorManagement.wErrorIdOffset;
	
ELSE
	bEventSendingOnceActive := TRUE;
	
	//Reset index in order to start scanning from the beginning
		iEvtSendingIndex := 0;
END_IF
END_METHOD

METHOD PRIVATE M_SendEvents		//Sends the Event for every SysErrror in the SysError List
VAR 
	i : UINT;
	localEvt : sSystemErrorEvent;
END_VAR
//Only Intervals above 100 ms (processing cycle)
IF tEventIntervalTime < T#100MS THEN
	tEventIntervalTime := T#100MS;
END_IF

//Sending

IF tEventIntervalTimer.Q THEN
	
	tEventIntervalTimer(IN := FALSE);
	
	FOR i := iEvtSendingIndex TO (ERROR_ARRAY_SIZE-1) DO
			IF SysErrorList[i].SysErrorMessageID <> 0 THEN //not empty	
														
					IF CurNotificationMode= eErrorNotificationMode.SENDING_ERRORS_ALWAYS_PERIODICALLY OR bEventSendingOnceActive THEN	
						//send every error
						M_CreateEvent(sysErr := SysErrorList[i]);		
						SysErrorList[i].bErrorWasSent		:= TRUE;
						tEventIntervalTimer(IN := TRUE);	
					
						// delete if it is a warning to prevent array overflow
						IF SysErrorList[i].ErrorMsg.ErrorTyp = eErrorTypes._WARNING THEN
							SysErrorList[i] := EMPTY_SYS_ERROR;
						END_IF
						
						EXIT;
						
					ELSIF CurNotificationMode = eErrorNotificationMode.SENDING_ERRORS_ONCE_IMMEDIATLY THEN
						
						IF NOT SysErrorList[i].bErrorWasSent THEN
							//send only errors which have not been sent before
							M_CreateEvent(sysErr := SysErrorList[i]);		
							SysErrorList[i].bErrorWasSent		:= TRUE;
							tEventIntervalTimer(IN := TRUE);								
							
							// delete if it is a warning to prevent array overflow
							IF SysErrorList[i].ErrorMsg.ErrorTyp = eErrorTypes._WARNING THEN
								SysErrorList[i] := EMPTY_SYS_ERROR;
							END_IF
														
							EXIT;
							
						END_IF
					END_IF
					
			END_IF		
	END_FOR
		
	iEvtSendingIndex := inc(i);
	
	IF iEvtSendingIndex >= ERROR_ARRAY_SIZE THEN
		iEvtSendingIndex := 0;
		bEventSendingOnceActive := FALSE;
	END_IF
	
ELSE
	tEventIntervalTimer(IN := TRUE, PT := tEventIntervalTime);
	
END_IF
END_METHOD

METHOD PUBLIC M_SendSingleError
VAR_INPUT
	iSysErrorMsgId : UINT;
END_VAR
VAR_OUTPUT
	bErrorMsgIdFound : 	BOOL := FALSE;
	bMethodError : 		BOOL := FALSE;
	MethodErrorMsg : 	sErrorMsg;
END_VAR
VAR
	sysErr : sSystemError;
	
END_VAR
sysErr := M_GetErrorInfo(	iSysErrorMsgID 	:= iSysErrorMsgId,
							bMethodError 	=> bMethodError,
							MethodErrorMsg 	=> MethodErrorMsg);
							
IF NOT bMethodError THEN
		M_CreateEvent(sysErr := sysErr);				
END_IF
END_METHOD

PROPERTY PUBLIC P_bHaveAllErrorsBeenSentAtLeastOnce : bool
GET
VAR
	i : UINT;
	bHaveAllBeenSend : BOOL := TRUE;;
END_VAR
FOR i := 0 TO (ERROR_ARRAY_SIZE - 1) DO
	IF SysErrorList[i].SysErrorMessageID <> 0 AND NOT SysErrorList[i].bErrorWasSent THEN
		bHaveAllBeenSend := FALSE;
		EXIT;
	END_IF
END_FOR

P_bHaveAllErrorsBeenSentAtLeastOnce := bHaveAllBeenSend;
END_GET
END_PROPERTY

PROPERTY PUBLIC P_ErrorNotificationMode : eErrorNotificationMode
GET
P_ErrorNotificationMode := CurNotificationMode;
END_GET
SET
CurNotificationMode := P_ErrorNotificationMode;
END_SET
END_PROPERTY

PROPERTY PUBLIC P_tEventIntervall : Time
GET
P_tEventIntervall := tEventIntervalTime;
END_GET
SET
tEventIntervalTime := P_tEventIntervall;
END_SET
END_PROPERTY

METHOD PRIVATE M_CreateEvent //Create an event from a system error object from array
VAR_INPUT
	sysErr : sSystemError;
END_VAR
VAR
	localEvt : sSystemErrorEvent;
END_VAR
//Prepare local evt structure				
	localEvt.SysErrorMessageID 		:= sysErr.SysErrorMessageID;
						
	localEvt.ErrorTyp 				:= sysErr.ErrorMsg.ErrorTyp;				
	localEvt.ErrorModuleId 			:= sysErr.ErrorMsg.wModule; 
	localEvt.ErrorCompId 			:= sysErr.ErrorMsg.wComponent;
	localEvt.ErrorId 				:= sysErr.ErrorMsg.wErrorNo;
	localEvt.iRelatedDocId			:= sysErr.ErrorMsg.iRelatedDocId;	
	
	IF NOT IsValidPtr(sysErr.ErrorMsg.pErrorHandler) THEN
		sysErr.ErrorMsg.pErrorHandler := ADR(ErrHand_Dummy);
		
	ELSE
			pErrHnd := sysErr.ErrorMsg.pErrorHandler;

	END_IF	 
		
	localEvt.AvailableHandlingModes := pErrHnd^.P_wAllowedHandlingModes;
	localEvt.EventChangeFlag 		:= switch(GVL_ErrorManagement.pEvt^.EventChangeFlag);
					
//Set final evt structure
	GVL_ErrorManagement.pEvt^ := localEvt;
END_METHOD

METHOD PRIVATE M_CreateLogData
VAR_INPUT
	pErr : sSystemError;
END_VAR
VAR
	sFuncName: STRING;
	strModule,
	strComp,
	strErrorId,
	strRelDocId,
	strErrorTyp,
	strLogMsg : STRING;
END_VAR
IF NOT GVL_ErrorManagement.bLoggingOnOff THEN
	RETURN;
END_IF

//Create log string
	strModule := CONCAT('|Module: ',WORD_TO_STRING(pErr.ErrorMsg.wModule));
	strLogMsg := CONCAT(strLogMsg, strModule);
	
	strComp := concat('|Component: ', WORD_TO_STRING(pErr.ErrorMsg.wComponent));
	strLogMsg := CONCAT(strLogMsg, strComp);
	
	strErrorId := concat('|ErrorId: ', WORD_TO_STRING(pErr.ErrorMsg.wErrorNo));
	strLogMsg := CONCAT(strLogMsg, strErrorId);
	
	strRelDocId := concat('|RelatedDocId: ', UDINT_TO_STRING(pErr.ErrorMsg.iRelatedDocId));
	strLogMsg := CONCAT(strLogMsg, strRelDocId);
	
	strErrorTyp := concat('|ErrorTyp: ', UINT_TO_STRING(pErr.ErrorMsg.ErrorTyp));
	strLogMsg := CONCAT(strLogMsg, strErrorTyp);

	sFuncName := pErr.ErrorMsg.sFunctionName;
	
//log data
CASE pErr.ErrorMsg.ErrorTyp OF
eErrorTypes._ERROR : 
						Logging.Error(Caller 	:= sFuncName, 
										Msg 	:= strLogMsg);	
										
eErrorTypes._FATAL : 
						Logging.Fatal(Caller 	:= sFuncName, 
										Msg 	:= strLogMsg);	
										
eErrorTypes._WARNING : 
						Logging.Warn(	Caller 	:= sFuncName, 
										Msg 	:= strLogMsg);	
ELSE
						Logging.Trace(Caller 	:= sFuncName, 
										Msg 	:= strLogMsg);	
END_CASE
END_METHOD

END_PROGRAM

// ErrorManagement/FB_ErrorHandler_Base
//{attribute 'hide_all_locals'}
FUNCTION_BLOCK FB_ErrorHandler_Base
VAR_INPUT
	bExecute: BOOL := FALSE;
END_VAR
VAR_OUTPUT
	bDone,
	bError : BOOL := FALSE;
END_VAR
VAR
	//Pre configuration
		iErrorIdToHandle 			: WORD := 0;	
	
		bAutomaticHandlingAllowed,
		bRepeatHandlingAllowed,
		bContinueHandlingAllowed 	: BOOL := FALSE;
	
	//Internal ariables - DO NOT OVERWRITE!
		iMethodHelpState : 	UINT := 0;
		bHandlerSet : 		BOOL := FALSE;
			
		HandlingModeSet :	eErrorHandlingMode;
		END_VAR



IF bExecute THEN	//Handler is executed
	IF bHandlerSet THEN
		
		CASE HandlingModeSet OF
			eErrorHandlingMode._AUTOMATIC : 	M_ExecuteHandling_Automatic();
			
			eErrorHandlingMode._REPEAT : 		M_ExecuteHandling_Repeat();
			
			eErrorHandlingMode._CONTINUE : 		M_ExecuteHandling_Continue();
			
		END_CASE
		
	ELSE
		bDone 	:= TRUE;
		bError 	:= TRUE; 
	END_IF
	
ELSE 				//Reset everything
	M_ResetFb();
	
END_IF

METHOD PUBLIC M_ExecuteHandling_Automatic
//to be overwritten in derived FB, if HandlingMode is activated
//iMethodHelpState can be used to create a method statemachine

//To following flags have to be set by the method
	bDone := TRUE;
	bError := TRUE;
END_METHOD

METHOD PUBLIC M_ExecuteHandling_Continue
//to be overwritten in derived FB, if HandlingMode is activated
//iMethodHelpState can be used to create a method statemachine

//To following flags have to be set by the method
	bDone := TRUE;
	bError := TRUE;
END_METHOD

METHOD PUBLIC M_ExecuteHandling_Repeat
//to be overwritten in derived FB, if HandlingMode is activated
//iMethodHelpState can be used to create a method statemachine

//To following flags have to be set by the method
	bDone := TRUE;
	bError := TRUE;
END_METHOD

METHOD PRIVATE M_IsHandlingModeAllowed : bool
VAR_INPUT
	HandlingModeToBeChecked :	eErrorHandlingMode;
END_VAR
VAR 
	bResult: BOOL:=FALSE;	
END_VAR
CASE HandlingModeToBeChecked OF
	eErrorHandlingMode._AUTOMATIC : 	bResult := bAutomaticHandlingAllowed;
	eErrorHandlingMode._REPEAT : 		bResult := bRepeatHandlingAllowed;
	eErrorHandlingMode._CONTINUE : 		bResult := bContinueHandlingAllowed;
	
ELSE
		bResult := FALSE;		 	
END_CASE

M_IsHandlingModeAllowed := bResult;
END_METHOD

METHOD PRIVATE M_ResetFb
bExecute 	:= FALSE;
bDone		:= false;
bError 		:= FALSE;
iMethodHelpState := 0;

bHandlerSet := FALSE;		
HandlingModeSet := eErrorHandlingMode._NONE;
END_METHOD

METHOD PUBLIC M_SetHandling
VAR_INPUT
	ErrorId 		: WORD;
	ErrHandlingMode : eErrorHandlingMode;
END_VAR
VAR_OUTPUT
	bMethodError 	: BOOL := FALSE;
	MethodErrorMsg 	: sErrorMsg;
END_VAR
MethodErrorMsg.wComponent 		:= GVL_ErrorManagement.wCompId;
MethodErrorMsg.sFunctionName 	:= 'M_HandleError';
MethodErrorMsg.wErrorNo 		:= GVL.ERR_NO_ERROR;

IF NOT THIS^.P_bHandlingAvailable THEN
	bMethodError := TRUE;
	MethodErrorMsg.wErrorNo 	:= GVL_ErrorManagement_ERROR_IDS.ERR_FSM_NO_ERROR_HANDLING_AVAILABLE_INSIDE_HANDLER + GVL_ErrorManagement.wErrorIdOffset;
	
ELSIF ErrorId <> iErrorIdToHandle THEN
	bMethodError := TRUE;
	MethodErrorMsg.wErrorNo 	:= GVL_ErrorManagement_ERROR_IDS.ERR_FSM_PRE_SET_HANDLER_ERRORID_DIFFERS + GVL_ErrorManagement.wErrorIdOffset;

ELSIF NOT M_IsHandlingModeAllowed(ErrHandlingMode) THEN
	bMethodError := TRUE;
	MethodErrorMsg.wErrorNo 	:= GVL_ErrorManagement_ERROR_IDS.ERR_FSM_ERROR_HANDLING_MODE_NOT_ALLOWED + GVL_ErrorManagement.wErrorIdOffset;
	
ELSE //No error, thus set flag to unlock handler execution
	M_ResetFb();
	
	HandlingModeSet	:= ErrHandlingMode;
	bHandlerSet 	:=TRUE;
	
END_IF
END_METHOD

PROPERTY PUBLIC P_bHandlingAvailable : bool
GET
P_bHandlingAvailable := (bAutomaticHandlingAllowed OR bRepeatHandlingAllowed or	bContinueHandlingAllowed);
END_GET
END_PROPERTY

PROPERTY PUBLIC P_wAllowedHandlingModes : word
GET
		P_wAllowedHandlingModes.0 := THIS^.P_bHandlingAvailable;
		P_wAllowedHandlingModes.1 := bAutomaticHandlingAllowed;
		P_wAllowedHandlingModes.2 := bRepeatHandlingAllowed;
		P_wAllowedHandlingModes.3 := bContinueHandlingAllowed;
END_GET
END_PROPERTY

END_FUNCTION_BLOCK

// Standard/Inc
FUNCTION Inc : uint //increment VAR "value" and return it 
VAR_IN_OUT
	value : UINT;
END_VAR

IF value >= 16#FFFF THEN
	value := 16#FFFF;
END_IF

value := value + 1;

Inc:= value;

END_FUNCTION

// Standard/IsValidPtr
FUNCTION IsValidPtr : bool
VAR_INPUT
	ptr : POINTER TO BYTE;
END_VAR

IsValidPtr :=  ptr <> 0;

END_FUNCTION

// Standard/Dec
FUNCTION Dec : uint //decrement VAR "value" and return it 
VAR_IN_OUT
	value : UINT;
END_VAR

IF value = 0 THEN
	value := 0;
END_IF

value := value - 1;

Dec := value;

END_FUNCTION

// AdsInterface/FB_wCMD_Handler_Base
//Author: 				Walther Ronny
//Version:				1.3
//Last change:			25.05.16
//See Release notes at the bottom
//{attribute 'hide_all_locals'}
{attribute 'reflection'}
FUNCTION_BLOCK PUBLIC FB_wCMD_Handler_Base				//Base Fb for handling of ADS communication of type TwRes and TwCmd
VAR_OUTPUT
    {attribute 'instance-path'}
    {attribute 'no_init'}
    sPath  	: STRING; 	//Instance path

END_VAR 
VAR_INPUT		
	Instanz: BYTE; 										//Instanz counter 
	pCmd : POINTER TO TxCmdRes;							//Pointer to incomming command structure from host
	pRes : POINTER TO TxCmdRes;							//Pointer to outgoing result structure from SPS
END_VAR
VAR	
	wCompId : WORD;		//Component ID
//Command configuration which has to be set by instantiated Fb - 	MUST !
	wVersion : 				WORD := 0;	//Expected version of incomming command
	iParTyp : 				BYTE := 0;	//Expected parameter type of incomming command, PAR_TYPE_REGARDLESS will switch test off
	iParCount : 			BYTE := 0;	//Expected parameter count of incomming command
	
//Command configuration which can be set by instantiated Fb - 	OPTIONALLY !
	bAbortionAllowed : 		BOOL 		:= FALSE;					//if yes, abortion from host is allowed all the time
	tExecutionTimeout : 	TIME 		:= ADS_EXECUTION_TIMEOUT; 	//Timeout while Execution running. T#0s equals off
	strInstanceName :		STRING(40);								//Name of instance of that base class (used only for logging purposes)
//Flag to indicate that the derived method "M_ExecuteCommand()" finished	
	bExecutionDone : BOOL := FALSE;	//flag to indicate that derived Execution is done				

//This variable can be used to hold the state of the derived M_ExecuteCommand() 
	iHelpState : UINT := 0;	//optional help variable to create a statemachine inside derive M_ExecuteCommand()
	
//Local Command and result structure objects - Will be read and written by base Fb and derived "M_ExecuteCommand()" method
	localRes: TwRes;
	localCmd: TwCmd;	
	
//Internal variables of base Fb - DO NOT CHANGE!	
	bCmdEnabledByExtern,								//Command is enabled/disabled  externally (by MainFSM)
	bCmdEnabledByIntern : 	BOOL:= TRUE;				//Command is enabled/disabled  internally during execution
		
	eState: eCmdProcessing := eCmdProcessing._RECEIVING;	//Current internal state of the base Fb		
	TimerExecutionTimeout : ton;						// Timer for Execution timeout
END_VAR
VAR CONSTANT
	//Command parameter types
	PAR_TYPE_REGARDLESS :		BYTE := 0;		//if this type is set, the parameter type will be not checked
	PAR_TYPE_ANSICHAR : 		BYTE := 16#41; //8bit
	PAR_TYPE_BYTE : 			BYTE := 16#42; //8bit
	PAR_TYPE_WIDECHAR : 		BYTE := 16#43; //16bit
	PAR_TYPE_FLOAT : 			BYTE := 16#44; //64bit	
	PAR_TYPE_SHORTINT : 		BYTE := 16#53; //8bit	
	PAR_TYPE_SMALLINT : 		BYTE := 16#4D; //16bit
	PAR_TYPE_LONGINT : 			BYTE := 16#49; //32bit
	PAR_TYPE_LONGWORD : 		BYTE := 16#4C; //32bit
	PAR_TYPE_WORD : 			BYTE := 16#57; //16bit
	PAR_TYPE_BIT : 				BYTE := 16#58;
	
	ADS_EXECUTION_TIMEOUT :		TIME := T#30S;		//Timeout while derived Execution method is executed. T#0S equals OFF

		// command
	cAbort:						WORD := 0;			// command abort				
	cRcv:						WORD := 1;			// command receive				
	cExec:						WORD := 2;			// command start				
	// result
	cIdle: 						WORD := 0;      	// not  defined					
	cRcvd:						WORD := 1;      	// command received 			
	cActive:					WORD := 2;			// command active started 		
	cFinOk:						WORD := 4;			// command finished ok			
	cFinAbrtd:					WORD := 5;			// command aborted				
	cFinErr:					WORD := 6;			// command finished error		
END_VAR

(*
Release notes:
1.0 First release. Tested on Holo machine in Munich. 25.01.16
1.1 Aborting modified and tested. Constants included in FB. 26.01.16
1.2 Bug M_ReceiveCommand PARTYP_REGARDLESS fixed
1.3 Walther Ronny, 25.05.16
	- Variable strInstanceName added
	- Method M_Log() added
	- Logging added
*)

//Create local copy of received command struct
	localCmd:=pCmd^.wCmd;

CASE eState OF
	
	eCmdProcessing._RECEIVING: 	//Receiving command
	
				//Check id, thus it might have been changed
					wCompId := GVL_AdsInterface.wCompId_IncomingAds;
				
				M_ReceiveCommand();
				
				IF localRes.Status = cRcvd THEN //was something received?	
					
					//Log data
						M_Log(	LogLevel 	:= eLogLevel.TRACE, 
								strMethod 	:= 'FB_wCMD_Handler_Base',
								strLogMsg 	:= '|ADS - command received from host');	
	
					eState := eCmdProcessing._WAITING_FOR_START;
					
				END_IF
				
	eCmdProcessing._WAITING_FOR_START:	//Waiting for Start from Host
	
				IF localCmd.Control = cExec THEN //check if the command was started by the host
					//Log data
						M_Log(	LogLevel 	:= eLogLevel.TRACE, 
								strMethod 	:= 'FB_wCMD_Handler_Base',
								strLogMsg 	:= '|ADS - command started by host');	
						
					IF localRes.Error = GVL.ERR_NO_ERROR THEN //Check if an error during receiving ocurred
						//Reset variables for derived "M_ExecuteCommand()" method	
							bExecutionDone := FALSE;
							iHelpState := 0;	
						
						localRes.Status := cActive;					
						eState := eCmdProcessing._EXECUTING;
						
						//start timeout timer
							TimerExecutionTimeout(IN := TRUE, PT := tExecutionTimeout);
					ELSE						
						eState := eCmdProcessing._FINISHING;
						
					END_IF
					
				END_IF
					
					
	eCmdProcessing._EXECUTING:	//Executing command
			
				IF bExecutionDone THEN //flag will be set by derived method if execution done									
					eState := eCmdProcessing._FINISHING; 
					
				ELSIF TimerExecutionTimeout.Q AND tExecutionTimeout <> T#0S THEN
					localRes.ErrorComp := wCompId;	
					localRes.Error := GVL_AdsInterface_ERROR_IDS.ERR_ITF_COMMAND_EXECUTION_TIMEOUT + GVL_AdsInterface.wErrorIdOffset_IncomingAds;
					
					eState := eCmdProcessing._FINISHING; 			
					
				ELSE //derived method will be executed
					M_ExecuteCommand();
						
				END_IF
	
		
	eCmdProcessing._FINISHING: //Finishing Command
		
				M_FinishCommand();
				
				//reset timer
					TimerExecutionTimeout.IN := FALSE;
				
				
	eCmdProcessing._ABORTING: //Aborting Command
				
				eState := eCmdProcessing._FINISHING; 
				
END_CASE

//check if aborted by host and command configured "bAbortionAllowed
//Note: 	Thus abortion is possible all the time the execution could be interuppted at an unsafe state!
//			Preferable abortion should be allowed only for service commands which a triggered manually from an operator.
	IF localCmd.Control = cAbort AND bAbortionAllowed 
		AND eState <> eCmdProcessing._ABORTING 		//Not allowed cause aborting already active
		AND eState <> eCmdProcessing._FINISHING 	//Not allowed cause command is finishing anyway
		AND eState <> eCmdProcessing._RECEIVING		//Not allowed cause command have not been started yet
		THEN 
			
			IF eState = eCmdProcessing._EXECUTING THEN  //cause eventually leaving unsafe state, throw error
				localRes.ErrorComp := wCompId;	
				localRes.Error := GVL_AdsInterface_ERROR_IDS.ERR_ITF_COMMAND_WAS_ABORTED_BY_HOST_DURING_EXECUTION + GVL_AdsInterface.wErrorIdOffset_IncomingAds;
				
			END_IF
			
			eState := eCmdProcessing._ABORTING;
			
	END_IF

TimerExecutionTimeout();
		
pRes^.wRes := localRes;

METHOD PUBLIC FINAL M_EnableCmd
VAR_INPUT
	bEnable : BOOL := FALSE; //TRUE = Command is enabled, FALSE = Command i disabled
END_VAR
bCmdEnabledByExtern := bEnable;
END_METHOD

METHOD PUBLIC M_ExecuteCommand // to be derived and customized....
// to be derived and customized....



//To DO`s of the derived Method:
 
//1. Check Data for correctness
//2. set optional result data 
//3. iHelpState vaiable can be used
//4. if an Error occured localRes.Error and localRes.ErrorComp has to be set!
//5. at last the "bExecutionDone" flag has to be set. This will start the transition to the M_FinishCommand Method inside the base FB.

